# B&R Automation Studio project NAINV104C00R8L515F00 (part 32)

#### Act_InitLocal.st - Do Not Change!!!
```iecst
(** 2021-08-01 **)
ACTION Act_InitLocal:

	//Input Reference Link To Local Variable
	p_eAct ACCESS ADR(eAct);
	p_udiRstErr ACCESS ADR(udiRstErr);
	p_bPrep ACCESS ADR(bPrep);
	p_bEn ACCESS ADR(bEn);
	p_bDis ACCESS ADR(bDis);
	p_tyParam ACCESS ADR(tyParam);
	p_sIPAddr ACCESS ADR(sIPAddr);
	pa_usiMacAddr ACCESS ADR(a_usiMacAddr);
	p_tyDTStructure ACCESS ADR(tyDTStructure);
	p_dtCurrDT ACCESS ADR(dtCurrDT);
	p_sMcId ACCESS ADR(sMcId);
	p_sMagazineId ACCESS ADR(sMagazineId);
	p_iSlotId ACCESS ADR(iSlotId);
	p_eBoardTransfer1 ACCESS ADR(eBoardTransfer1);
	p_eBoardTransfer2 ACCESS ADR(eBoardTransfer2);
	p_eBoardTransfer3 ACCESS ADR(eBoardTransfer3);
	p_eBoardTransfer4 ACCESS ADR(eBoardTransfer4);
	p_sVersion ACCESS ADR(sVersion);
	p_sBarcode ACCESS ADR(sBarcode);
	p_sRecipeNm ACCESS ADR(sRecipeNm);
	p_udiSndBffrSize ACCESS ADR(udiSndBffrSize);
	p_udiRcvBffrSize ACCESS ADR(udiRcvBffrSize);
	p_udiAliveIdleTimeInSec ACCESS ADR(udiAliveIdleTimeInSec);
	p_tConnTimeOut ACCESS ADR(tConnTimeOut);
	p_diTransferInTO ACCESS ADR(diTransferInTO);
	p_bNewBrdAvlLastZone ACCESS ADR(bNewBrdAvl);
	p_bOpsRun ACCESS ADR(bOpsRun);
	p_udiFileKeepDay ACCESS ADR(udiFileKeepDay);
	p_sConfigFileName ACCESS ADR(sConfigFileName);
	p_sProgNm ACCESS ADR(sProgNm);
	p_bNtSettingsLoadDone ACCESS ADR(bNtSettingsLoadDone);
	p_bSvyPrep ACCESS ADR(bSvyPrep);
	p_bSvyEn ACCESS ADR(bSvyEn);
	p_bQueryWorkOrderInfo ACCESS ADR(bQueryWorkOrderInfo);
	p_bReinsertBrd ACCESS ADR(bReinsertBrd);
	p_tyHermesConfiguration ACCESS ADR(tyHermesCurrConfiguration);
	p_bUSHermesStopTransport1 ACCESS ADR(bUSHermesStopTransportSnd1); //Lane 1
	p_bUSHermesStopTransport2 ACCESS ADR(bUSHermesStopTransportSnd2); //Lane 2
	p_bUSHermesStopTransport3 ACCESS ADR(bUSHermesStopTransportSnd3); //Lane 3
	p_bUSHermesStopTransport4 ACCESS ADR(bUSHermesStopTransportSnd4); //Lane 4
	p_tyUSBoardArrived1 ACCESS ADR(tyUSHermesBoardArrivedData1); //Lane 1
	p_tyUSBoardArrived2 ACCESS ADR(tyUSHermesBoardArrivedData2); //Lane 2
	p_tyUSBoardArrived3 ACCESS ADR(tyUSHermesBoardArrivedData3); //Lane 3
	p_tyUSBoardArrived4 ACCESS ADR(tyUSHermesBoardArrivedData4); //Lane 4
	p_bDSHermesTransportFinished1 ACCESS ADR(bDSHermesTransportFinishedSnd1); //Lane 1
	p_bDSHermesTransportFinished2 ACCESS ADR(bDSHermesTransportFinishedSnd2); //Lane 2
	p_bDSHermesTransportFinished3 ACCESS ADR(bDSHermesTransportFinishedSnd3); //Lane 3
	p_bDSHermesTransportFinished4 ACCESS ADR(bDSHermesTransportFinishedSnd4); //Lane 4
	p_tyDSBoardDeparted1 ACCESS ADR(tyDSHermesBoardDepartedData1); //Lane 1
	p_tyDSBoardDeparted2 ACCESS ADR(tyDSHermesBoardDepartedData2); //Lane 2
	p_tyDSBoardDeparted3 ACCESS ADR(tyDSHermesBoardDepartedData3); //Lane 3
	p_tyDSBoardDeparted4 ACCESS ADR(tyDSHermesBoardDepartedData4); //Lane 4
	p_sInfoMsg ACCESS ADR(sInfoMsg);
	p_sInfoMsg1 ACCESS ADR(sInfoMsg1);
	p_sInfoMsg2 ACCESS ADR(sInfoMsg2);
	p_sInfoMsg3 ACCESS ADR(sInfoMsg3);
	p_sInfoMsg4 ACCESS ADR(sInfoMsg4);
	p_sInfoMsg5 ACCESS ADR(sInfoMsg5);
	p_sInfoMsg6 ACCESS ADR(sInfoMsg6);
	p_bInternalUse ACCESS ADR(bInternalUse);
	p_sInternalRcv ACCESS ADR(sInternalRcv);
	p_bAcceptCondition ACCESS ADR(bAcceptCondition);
	p_bAllZonesEmpty ACCESS ADR(bAllZonesEmpty);
	p_bDeleteWorkOrder ACCESS ADR(bDeleteWorkOrder);
	p_bFirstMcIntheLine ACCESS ADR(bFirstMcIntheLine);
	p_sRetainFileName ACCESS ADR(sRetainFileName);
	p_udiRetainDataAddr ACCESS ADR(udiRetainDataAddr);
	p_udiRetainDataLen ACCESS ADR(udiRetainDataLen);

END_ACTION
```

#### Act_Initial.st - Do Not Change!!!
```iecst
(** 2021-08-01 **)
ACTION Act_Initial:

	//Initial
	sStatTxt	:= a_sStatText[eStat];

	fbCreateSvr.udiSndBffrSize		:= p_udiSndBffrSize;
	fbCreateSvr.udiRcvBffrSize		:= p_udiRcvBffrSize;
	fbCreateSvr.udiAliveIdleTmInSec	:= p_udiAliveIdleTimeInSec;
	fbCreateSvr(bEn := FALSE);

	fbListen(bEn := FALSE);

	fbRcv.udiBffrSize	:= SIZEOF(sRcv);
	fbRcv.p_BffrDest	:= ADR(sRcv);
	fbRcv(bEn := FALSE);

	fbSend.p_BffrDest	:= ADR(sSnd);
	fbSend(bEn := FALSE);

	fbCloseSvr(bEn := FALSE);
	fbCloseClnt(bEn := FALSE);

	fbParseXMLTable.p_XMLTable	:= ADR(a_tyXMLTableDataRcv);

	fbCheckAlive(bEn := FALSE);

	fbCheckAliveSendPing(bEn := FALSE);

	fbCheckAliveRcvPing(bEn := FALSE);

	fbSequenceSvy.p_tyMsgTypeRcv	:= ADR(tyMsgTypeRcv);
	fbSequenceSvy(bEn := FALSE);

	fbSequenceTO(bEn := FALSE);

	fbFileAppend1.sDevice	:= 'Log';
	fbFileAppend1(bEn := FALSE);

	fbFileOldDel1.sDevice			:= 'Log';
	fbFileOldDel1.sPath				:= '';
	fbFileOldDel1.sKeyword			:= p_sProgNm;
	fbFileOldDel1.udiFileKeepDay	:= p_udiFileKeepDay;
	fbFileOldDel1(bEn := FALSE);

	fbFileRead1.sDevice			:= 'Retain';
	fbFileRead1.sFile			:= p_sRetainFileName;
	fbFileRead1.udiOffset		:= 0;
	fbFileRead1(bEn := FALSE);

	fbFileWrite1.sDevice		:= 'Retain';
	fbFileWrite1.sFile			:= p_sRetainFileName;
	fbFileWrite1.udiOffset		:= 0;
	fbFileWrite1.udiOption		:= 0;
	fbFileWrite1(bEn := FALSE);

END_ACTION
```

#### Act_Main.st - Do Not Change!!!
```iecst
(** 2021-08-01 **)
ACTION Act_Main:

	IF eStatOld <> eStat THEN
		fbFileOldDel1(bEn := FALSE);
		fbFileRead1(bEn := FALSE);
		fbFileWrite1(bEn := FALSE);
		bFileNotFound	:= FALSE;
		sStatTxt	:= a_sStatText[eStat];

		eStatOld	:= eStat;

		eStatus		:= Busy;
	END_IF

	//Main
	CASE eStat OF

		HermesActIdle:
			eStatus	:= Idle;

		HermesActBGStartRun:
			IF eStatus = Idle OR eStatus = Busy THEN

				bRun	:= TRUE;
				bStop	:= FALSE;
				eStatus	:= Done;

			END_IF

		HermesActBGStopRun:
			IF eStatus = Idle OR eStatus = Busy THEN

				bStop	:= TRUE;
				eStatus	:= Done;

			END_IF

		HermesActDeleteOldLog:
			IF eStatus = Idle OR eStatus = Busy THEN

				eStatus	:= Busy;

				fbFileOldDel1.dtDTNow	:= p_dtCurrDT;
				fbFileOldDel1(bEn := TRUE);
				IF fbFileOldDel1.udiStatus = 0 THEN
					eStatus	:= Done;
				ELSIF fbFileOldDel1.udiStatus < 65534 THEN
					eStatus		:= Error;

					IF fbFileOldDel1.udiStatus = 1910 THEN
						udiStatus	:= 10111;	//Get Directory Info Error While Deleting Old Log
					ELSIF fbFileOldDel1.udiStatus = 1911 THEN
						udiStatus	:= 10112;	//Directory Read Error While Deleting Old Log
					ELSIF fbFileOldDel1.udiStatus = 1912 THEN
						udiStatus	:= 10113;	//File Delete Error While Deleting Old Log
					ELSE
						udiStatus	:= fbFileOldDel1.udiStatus;
					END_IF
				END_IF

			END_IF

		HermesActReadRetain:
			IF eStatus = Idle OR eStatus = Busy THEN

				eStatus	:= Busy;

				fbFileRead1.p_Dest	:= p_udiRetainDataAddr;
				fbFileRead1.udiLen	:= p_udiRetainDataLen;
				fbFileRead1(bEn := TRUE);

				IF fbFileRead1.udiStatus = 0 THEN
					eStatus	:= Done;
				ELSIF fbFileRead1.udiStatus < 65534 THEN
					eStatus	:= Error;

					IF fbFileRead1.udiStatus = 1900 THEN
						udiStatus	:= 10114;	//File Open Error While Reading Retain File
					ELSIF fbFileRead1.udiStatus = 1902 THEN
						udiStatus	:= 10115;	//File Read Error While Reading Retain File
					ELSIF fbFileRead1.udiStatus = 1904 THEN
						udiStatus	:= 10116;	//File Close Error While Reading Retain File
					ELSIF fbFileRead1.udiStatus = 1915 THEN
						eStatus			:= Done;
						bFileNotFound	:= TRUE;
					ELSE
						udiStatus	:= fbFileRead1.udiStatus;
					END_IF
				END_IF

			END_IF

		HermesActWriteRetain:
			IF eStatus = Idle OR eStatus = Busy THEN

				eStatus	:= Busy;

				fbFileWrite1.p_Src	:= p_udiRetainDataAddr;
				fbFileWrite1.udiLen	:= p_udiRetainDataLen;
				fbFileWrite1(bEn := TRUE);

				IF fbFileWrite1.udiStatus = 0 THEN
					eStatus	:= Done;
				ELSIF fbFileWrite1.udiStatus < 65534 THEN
					eStatus	:= Error;

					IF fbFileWrite1.udiStatus = 1900 THEN
						udiStatus	:= 10117;	//File Open Error While Writing Retain File
					ELSIF fbFileWrite1.udiStatus = 1901 THEN
						udiStatus	:= 10118;	//File Create Error While Writing Retain File
					ELSIF fbFileWrite1.udiStatus = 1903 THEN
						udiStatus	:= 10119;	//File Write Error While Writing Retain File
					ELSIF fbFileWrite1.udiStatus = 1904 THEN
						udiStatus	:= 10120;	//File Close Error While Writing Retain File
					ELSIF fbFileWrite1.udiStatus = 1914 THEN
						udiStatus	:= 10121;	//Directory Does Not Exist While Writing Retain File
					ELSE
						udiStatus	:= fbFileWrite1.udiStatus;
					END_IF
				END_IF

			END_IF

		ELSE
			IF eStatus = Idle OR eStatus = Busy THEN
				eStatus	:= Done;
			END_IF

	END_CASE

END_ACTION
```

#### Act_Background.st - Do Not Change!!!
```iecst
(** 2021-08-01 **)
ACTION Act_Background:

	IF bRun = TRUE THEN
		IF udiSvrIdent = 0 THEN
			IF p_bInternalUse = FALSE THEN
				Act_Background_TCPCreateSvr;

				tyParamOld	:= p_tyParam;
			ELSE
				udiSvrIdent	:= 1;
			END_IF

		ELSE
			IF bRstConnection = FALSE THEN

				Act_Background_ChgConfig;

				IF udiClntIdent = 0 THEN
					IF p_bInternalUse = FALSE THEN
						Act_Background_TCPListen;
					ELSE
						udiClntIdent	:= 1;
					END_IF

				ELSE
					Act_Background_TCPRcv;

					Act_Background_NotificationRcv;

					Act_Background_IllegalMsg;
					Act_Background_ChkParamRcv;
					Act_Background_CmpParamRcv;
					Act_Background_UpdtConfig;

					IF bHandshakeDone = TRUE THEN
						IF (p_tyParam.tSndAlive <> T#0s) AND (p_tyParam.tRcvAlive <> T#0s) THEN
							IF tySServiceDescriptionRcv.tyData.tySupportedFeatures.bFeatureCheckAliveResponse = TRUE AND p_tyParam.bFeatureCheckAliveResponse = TRUE THEN
								Act_Background_ChkAliveSendPing;
								Act_Background_ChkAliveRcvPing;
							ELSE
								Act_Background_ChkAlive;
							END_IF
						ELSE
							fbCheckAlive(bEn := FALSE);
							fbCheckAliveSendPing(bEn := FALSE);
							fbCheckAliveRcvPing(bEn := FALSE);
						END_IF
					END_IF

					Act_Background_Sequence;
					Act_Background_SequenceTO;
					Act_Background_Err;

					IF tySServiceDescriptionRcv.tyAvl.tySupportedFeatures.bFeatureSendWorkOrderInfo = TRUE AND (p_tyParam.bFeatureQueryWorkOrderInfo OR p_bHermesReinsertBoard) AND bHandshakeDone THEN
						Act_Background_QueryWorkOrderInfo;
					END_IF

					Act_Background_SendBoardArrivedLane1;
					Act_Background_SendBoardArrivedLane2;
					Act_Background_SendBoardArrivedLane3;
					Act_Background_SendBoardArrivedLane4;
					Act_Background_SendBoardDepartedLane1;
					Act_Background_SendBoardDepartedLane2;
					Act_Background_SendBoardDepartedLane3;
					Act_Background_SendBoardDepartedLane4;
					Act_Background_TCPSend;

					Act_Background_Log;

				END_IF

			ELSE
				IF udiClntIdent <> 0 THEN
					Act_Background_TCPCloseClnt;
				ELSE
					IF udiSvrIdent <> 0 THEN
						Act_Background_TCPCloseSvr;
					END_IF
				END_IF

			END_IF

			//Second Client Connected
			IF udiClntIdentExtra = 0 THEN

			ELSE

			END_IF

		END_IF

		Act_Background_Stop;

	END_IF

	IF EDGENEG(bRun) OR EDGENEG(udiSvrIdent = 0) THEN
		//Reset
		fbCreateSvr(bEn := FALSE);
	END_IF

	IF EDGENEG(bRun) OR EDGENEG(udiClntIdent = 0) THEN
		//Reset
		fbListen(bEn := FALSE);

		bConnected	:= bRun;
	END_IF

	IF EDGENEG(bRun) OR EDGENEG(udiSvrIdent <> 0) OR EDGENEG(udiClntIdent <> 0) THEN
		fbRcv(bEn := FALSE);
		fbSequenceSvy(bEn := FALSE);
		fbSequenceTO(bEn := FALSE);
		fbCheckAlive(bEn := FALSE);
		fbCheckAliveSendPing(bEn := FALSE);
		fbCheckAliveRcvPing(bEn := FALSE);
		fbSend(bEn := FALSE);

		fbFileAppend1(bEn := FALSE);
		iWriteLogStep	:= 0;

		bConnected		:= FALSE;
		bHandshakeDone	:= FALSE;
		bRstState		:= FALSE;

		memset(ADR(tyMsgTypeRcv) , 0 , SIZEOF(tyMsgTypeRcv));
		memset(ADR(a_eMsgSend) , 0 , SIZEOF(a_eMsgSend));
		udiMsgSendBffr	:= 0;
	END_IF

	IF EDGENEG(bRun) OR EDGENEG(udiSvrIdent <> 0) THEN
		bRstConnection	:= FALSE;
		fbCloseSvr(bEn := FALSE);
	END_IF

	IF EDGENEG(bRun) OR EDGENEG(udiClntIdent <> 0) THEN
		fbCloseClnt(bEn := FALSE);
	END_IF

	//Reset Error
	IF (eStatus1 = Error) AND bRstErr THEN
		eStatus1	:= Idle;
		udiStatus1	:= 0;

		fbCreateSvr(bEn := FALSE);
		fbListen(bEn := FALSE);
		fbRcv(bEn := FALSE);
		fbSequenceSvy(bEn := FALSE);
		fbSend(bEn := FALSE);
		fbCloseSvr(bEn := FALSE);
		fbCloseClnt(bEn := FALSE);
		fbCheckAlive(bEn := FALSE);
		fbCheckAliveSendPing(bEn := FALSE);
		fbCheckAliveRcvPing(bEn := FALSE);
		fbSequenceTO(bEn := FALSE);

		fbFileAppend1(bEn := FALSE);
		iWriteLogStep	:= 0;

		bConnected		:= FALSE;
		bHandshakeDone	:= FALSE;
		bRstConnection	:= FALSE;
		bRstState		:= FALSE;

		memset(ADR(tyMsgTypeRcv) , 0 , SIZEOF(tyMsgTypeRcv));
		memset(ADR(a_eMsgSend) , 0 , SIZEOF(a_eMsgSend));
		udiMsgSendBffr	:= 0;
	END_IF

	IF (eStatus2 = Error) AND bRstErr THEN
		eStatus2	:= Idle;
		udiStatus2	:= 0;

		fbSequenceTO(bEn := FALSE);

	END_IF

	IF (eStatus3 = Error) AND bRstErr THEN
		eStatus3	:= Idle;
		udiStatus3	:= 0;

		fbFileAppend1(bEn := FALSE);
		iWriteLogStep	:= 0;
	END_IF

END_ACTION
```

#### Act_Background_ProcessData.st - Do Not Change!!!
```iecst
(** 2021-08-01 **)
ACTION Act_Background_ProcessData:

	//Write Config into "Hermes"
	fbDelayTm(IN := bWriteConfig, PT := T#0.5S); //Small Delay 0.5s to let Hermes take the Data, before WriteConfig

	IF fbDelayTm.Q THEN

		eHermesAct := HermesActWriteConfig;
		eMcParamAct := McParamActWrite;

		IF p_eHermesStatus = Done AND p_eHermesStat = HermesActWriteConfig AND p_eMcParamStat = McParamActWrite AND p_eMcParamStatus = Done THEN

		eMcParamAct     := McParamActIdle;
	   	eHermesAct		:= HermesActIdle;
		bWriteConfig    := FALSE;
		bUpdateUIData   := TRUE;
		fbDelayTm(IN := FALSE);
		tyInfoData.sProgNm		:= p_sProgNm;
		tyInfoData.udiCode		:= 10000;
		tyInfoData.eSeverity	:= AlmSeverityInfo;
		tyInfoData.sAlmMsg		:= p_sInfoMsg;

	    ELSIF  (p_eHermesStatus = Error AND p_eHermesStat = HermesActWriteConfig) OR (p_eMcParamStat = McParamActWrite AND p_eMcParamStatus = Error)  THEN

			eMcParamAct     := McParamActIdle;
		    eHermesAct		:= HermesActIdle;
		    bWriteConfig    := FALSE;
		    bUpdateUIData   := FALSE;
			fbDelayTm(IN := FALSE);

			fHermesAddOneMsgSend(ADR(a_eMsgSend) , ADR(udiMsgSendBffr) , HermesMsgTypeNotification);

			udiStatus2 := 10199; //SetConfiguration Failed, Please Send Again
			tyNotificationSnd.tyAvl.bSeverity			:= TRUE;
			tyNotificationSnd.tyAvl.bNotificationCode	:= TRUE;
			tyNotificationSnd.tyAvl.bDescription		:= TRUE;
			tyNotificationSnd.tyData.eSeverity			:= HermesSeverityFatalError;
			tyNotificationSnd.tyData.iNotificationCode	:= UDINT_TO_INT(udiStatus2);
			tyNotificationSnd.tyData.sDescription		:= a_tyAlmText[udiStatus2].sAlmText;

		END_IF
	END_IF

	//Update UI
	IF bUpdateUIData THEN
		tyInfoData.sProgNm		:= p_sProgNm;
		tyInfoData.udiCode		:= 10000;
		tyInfoData.eSeverity	:= AlmSeverityInfo;
		tyInfoData.sAlmMsg		:= p_sInfoMsg;
	END_IF

	//Auto Reset
	fbDelayTm1(IN := bUpdateUIData , PT := T#2S); //Auto reset the Info Msg C0009 page. No need press.
	IF fbDelayTm1.Q = TRUE THEN

		//Clear Info Message
		tyInfoData.sProgNm		:= '';
		tyInfoData.udiCode		:= 0;
		tyInfoData.eSeverity	:= AlmSeverityNA;
		tyInfoData.sAlmMsg		:= '';

		bUpdateUIData  := FALSE;
		bFoundIndexUS1 := FALSE;
		bFoundIndexUS2 := FALSE;
		bFoundIndexUS3 := FALSE;
		bFoundIndexUS4 := FALSE;
		bFoundIndexDS1 := FALSE;
		bFoundIndexDS2 := FALSE;
		bFoundIndexDS3 := FALSE;
		bFoundIndexDS4 := FALSE;

		fbDelayTm1(IN := FALSE);
	END_IF

	//BatchId from Supervisory System
	sBatchId := tySendWorkOrderInfoAcc.tyData.sBatchId;

	//Retain sWorkOrderId for machine power cycle
	p_udiRetainDataAddr	:= ADR(sWorkOrderId);
	p_udiRetainDataLen	:= SIZEOF(sWorkOrderId);

	//Write Retain
	IF EDGEPOS(bRcvWorkOrderInfo1) THEN
    	sWorkOrderId := tySendWorkOrderInfoAcc.tyData.sWorkOrderId; //Receive from Svy
		p_eAct := HermesActWriteRetain;

	ELSIF EDGENEG(p_bSvyEn = TRUE) OR EDGENEG(p_bSvyPrep = TRUE) THEN
		sWorkOrderId := ''; //Empty if Supervisory Hermes disable
		p_eAct := HermesActWriteRetain;

	ELSIF EDGENEG(p_tyHermesConfiguration.tySvyParam.bFeatureQueryWorkOrderInfo = TRUE) THEN
		sWorkOrderId := ''; //Empty if no support
		p_eAct := HermesActWriteRetain;

	ELSIF EDGEPOS(p_bDeleteWorkOrder) THEN
		sWorkOrderId := ''; //Delete from UI
		p_eAct := HermesActWriteRetain;
		p_bDeleteWorkOrder := FALSE;
	END_IF

	IF eStatus = Done AND eStat = HermesActWriteRetain THEN
		p_eAct		:= HermesActIdle;
	END_IF

//	//Testing -> Read Retain
//	IF EDGEPOS(bTest) THEN
//		p_eAct := HermesActReadRetain;
//	END_IF
//
//	IF eStatus = Done AND eStat = HermesActReadRetain THEN
//		p_eAct		:= HermesActIdle;
//	END_IF

	IF EDGEPOS(bTest) THEN

	END_IF

END_ACTION
```

#### Act_Background_TCPCreateSvr.st - Do Not Change!!!
```iecst
(** 2021-08-01 **)
ACTION Act_Background_TCPCreateSvr:

	IF eStatus1 <> Error THEN

		//Create Server
		fbCreateSvr.sSvrIP				:= p_sIPAddr;
		fbCreateSvr.uiSvrPort			:= p_tyParam.uiSvySvstemPort;
		fbCreateSvr(bEn := TRUE);

		IF fbCreateSvr.udiStatus = 0 THEN
			udiSvrIdent	:= fbCreateSvr.udiTCPIdent;
			fbCreateSvr(bEn := FALSE);

		ELSIF fbCreateSvr.udiStatus < 65534 THEN
			eStatus1	:= Error;

			IF fbCreateSvr.udiStatus = 2300 THEN
				udiStatus1	:= 10000;	//Invalid Ident While Creating Server
			ELSIF fbCreateSvr.udiStatus = 2302 THEN
				udiStatus1	:= 10001;	//Setting Keep Alive Interval Time Error While Creating Server
			ELSIF fbCreateSvr.udiStatus = 2303 THEN
				udiStatus1	:= 10002;	//Setting Keep Alive Idle Time Error While Creating Server
			ELSIF fbCreateSvr.udiStatus = 2304 THEN
				udiStatus1	:= 10003;	//Setting Keep Alive Count Error While Creating Server
			ELSIF fbCreateSvr.udiStatus = 2305 THEN
				udiStatus1	:= 10004;	//Setting Keep Alive Error While Creating Server
			ELSIF fbCreateSvr.udiStatus = 2306 THEN
				udiStatus1	:= 10005;	//Setting Receive Buffer Error While Creating Server
			ELSIF fbCreateSvr.udiStatus = 2307 THEN
				udiStatus1	:= 10006;	//Setting Send Buffer Error While Creating Server
			ELSIF fbCreateSvr.udiStatus = 2308 THEN
				udiStatus1	:= 10007;	//Setting No Waiting Error While Creating Server
			ELSIF fbCreateSvr.udiStatus = 2309 THEN
				udiStatus1	:= 10008;	//TCP Open Port Error While Creating Server
			ELSIF fbCreateSvr.udiStatus = 2310 THEN
				udiStatus1	:= 10009;	//Closing TCP Error While Creating Server
			ELSE
				udiStatus1	:= fbCreateSvr.udiStatus;
			END_IF

		END_IF

	END_IF

END_ACTION
```

#### Act_Background_TCPListen.st - Do Not Change!!!
```iecst
(** 2021-08-01 **)
ACTION Act_Background_TCPListen:

	IF eStatus1 <> Error AND eStatus2 <> Error THEN

		fbListen.udiSvrIdent	:= udiSvrIdent;
		fbListen(bEn := TRUE);

		IF fbListen.udiStatus = 0 THEN
			udiClntIdent	:= fbListen.udiClntIdent;
			fbListen(bEn := FALSE);

		ELSIF fbListen.udiStatus = 2311 THEN //No Client Connected
			fbListen(bEn := FALSE);

		ELSIF fbListen.udiStatus = 2312 OR (bConnected=FALSE) THEN
			udiStatus4	:= 10012;	//Supervisory Hermes Connection Lost
			fbListen(bEn := FALSE); //add

		ELSIF fbListen.udiStatus < 65534 THEN
			eStatus1	:= Error;

			IF fbListen.udiStatus = 2300 THEN
				udiStatus1	:= 10010;	//Invalid Ident While Listening Client
			ELSE
				udiStatus1	:= fbListen.udiStatus;
			END_IF

		END_IF

	END_IF

END_ACTION
```

#### Act_Background_TCPRcv.st - Do Not Change!!!
```iecst
(** 2020-10-20 **)
ACTION Act_Background_TCPRcv:

	IF eStatus1 <> Error THEN

		//Receive Data
		IF p_bInternalUse = FALSE THEN
			fbRcv.udiTCPIdent	:= udiClntIdent;
			fbRcv(bEn := TRUE);
		ELSE
			sRcv	:= p_sInternalRcv;
		END_IF

		IF (fbRcv.udiStatus = 0) OR ((p_bInternalUse = TRUE) AND (LEN(sRcv) > 0)) THEN

			fLogDTConvert(ADR(sDT) , p_dtCurrDT);
			memset(ADR(a_sLogList[udiLogCntr]) , 0 , SIZEOF(a_sLogList[udiLogCntr]));
			memcpy(ADR(a_sLogList[udiLogCntr]) + LEN(a_sLogList[udiLogCntr]) , ADR(sDT) , LEN(sDT));
			memcpy(ADR(a_sLogList[udiLogCntr]) + LEN(a_sLogList[udiLogCntr]) , ADR('$r$n') , LEN('$r$n'));
			memcpy(ADR(a_sLogList[udiLogCntr]) + LEN(a_sLogList[udiLogCntr]) , ADR('RCV_FRM_SVY$r$n') , LEN('RCV_FRM_SVY$r$n'));
			memcpy(ADR(a_sLogList[udiLogCntr]) + LEN(a_sLogList[udiLogCntr]) , ADR(sRcv) , LEN(sRcv));
			memcpy(ADR(a_sLogList[udiLogCntr]) + LEN(a_sLogList[udiLogCntr]) , ADR('$r$n$r$n') , LEN('$r$n$r$n'));

			udiLogCntr	:= udiLogCntr + 1;
			IF udiLogCntr = 11 THEN
				udiLogCntr	:= 1;
			END_IF

			fXMLConvertToTable(ADR(sRcv) , LEN(sRcv) , ADR(a_tyXMLTableDataRcv) , ADR(a_tyXMLTableDataRcv[0].sTitle) , SIZEOF(a_tyXMLTableDataRcv[0].sTitle) , ADR(a_tyXMLTableDataRcv[0].sValue) , SIZEOF(a_tyXMLTableDataRcv[0].sValue) , ADR(a_tyXMLTableDataRcv[0].uiSize) , SIZEOF(a_tyXMLTableDataRcv[0]) , SIZEOF(a_tyXMLTableDataRcv) / SIZEOF(a_tyXMLTableDataRcv[0]) , ADR(udiXMLTableWriteIdx));

			fbParseXMLTable.iTotalIdxWrite	:= UDINT_TO_INT(udiXMLTableWriteIdx);
			fbParseXMLTable;

			IF fbParseXMLTable.tyMsgType.bCheckAlive = TRUE THEN
				tyMsgTypeRcv.bCheckAlive	:= TRUE;
				tyCheckAliveRcv				:= fbParseXMLTable.tyCheckAlive;
			END_IF

			IF fbParseXMLTable.tyMsgType.bCheckAlivePing = TRUE THEN
				tyMsgTypeRcv.bCheckAlivePing	:= TRUE;
				tyCheckAlivePingRcv				:= fbParseXMLTable.tyCheckAlivePing;
			END_IF

			IF fbParseXMLTable.tyMsgType.bCheckAlivePong = TRUE THEN
				tyMsgTypeRcv.bCheckAlivePong	:= TRUE;
				tyCheckAlivePongRcv				:= fbParseXMLTable.tyCheckAlivePong;
			END_IF

			IF fbParseXMLTable.tyMsgType.bServiceDescription = TRUE THEN
				tyMsgTypeRcv.bServiceDescription	:= TRUE;
				tyServiceDescriptionRcv				:= fbParseXMLTable.tyServiceDescription;
			END_IF

			IF fbParseXMLTable.tyMsgType.bSServiceDescription = TRUE THEN
				tyMsgTypeRcv.bSServiceDescription	    := TRUE;
				tySServiceDescriptionRcv				:= fbParseXMLTable.tySServiceDescription;
			END_IF

			IF fbParseXMLTable.tyMsgType.bNotification = TRUE THEN
				tyMsgTypeRcv.bNotification	:= TRUE;
				tyNotificationRcv			:= fbParseXMLTable.tyNotification;
			END_IF

			IF fbParseXMLTable.tyMsgType.bBoardAvailable = TRUE THEN
				tyMsgTypeRcv.bBoardAvailable	:= TRUE;
				tyBoardAvailableRcv				:= fbParseXMLTable.tyBoardAvailable;

			END_IF

			IF fbParseXMLTable.tyMsgType.bRevokeBoardAvailable = TRUE THEN
				tyMsgTypeRcv.bRevokeBoardAvailable	:= TRUE;
			END_IF

			IF fbParseXMLTable.tyMsgType.bMachineReady = TRUE THEN
				tyMsgTypeRcv.bMachineReady	:= TRUE;
				tyMachineReady				:= fbParseXMLTable.tyMachineReady;
			END_IF

			IF fbParseXMLTable.tyMsgType.bRevokeMachineReady = TRUE THEN
				tyMsgTypeRcv.bRevokeMachineReady	:= TRUE;
			END_IF

			IF fbParseXMLTable.tyMsgType.bStartTransport = TRUE THEN
				tyMsgTypeRcv.bStartTransport	:= TRUE;
				tyStartTransport				:= fbParseXMLTable.tyStartTransport;
			END_IF

			IF fbParseXMLTable.tyMsgType.bStopTransport = TRUE THEN
				tyMsgTypeRcv.bStopTransport	:= TRUE;
				tyStopTransport				:= fbParseXMLTable.tyStopTransport;
			END_IF

			IF fbParseXMLTable.tyMsgType.bTransportFinished = TRUE THEN
				tyMsgTypeRcv.bTransportFinished	:= TRUE;
				tyTransportFinished				:= fbParseXMLTable.tyTransportFinished;
			END_IF

			IF fbParseXMLTable.tyMsgType.bSetConfiguration = TRUE THEN
				tyMsgTypeRcv.bSetConfiguration	:= TRUE;
				tySetConfigurationRcv			:= fbParseXMLTable.tySetConfiguration;
			END_IF

			IF fbParseXMLTable.tyMsgType.bGetConfiguration = TRUE THEN
				tyMsgTypeRcv.bGetConfiguration	:= TRUE;
			END_IF

			IF fbParseXMLTable.tyMsgType.bCurrentConfiguration = TRUE THEN
				tyMsgTypeRcv.bCurrentConfiguration	:= TRUE;
				tyCurrentConfigurationRcv			:= fbParseXMLTable.tyCurrentConfiguration;
			END_IF

			IF fbParseXMLTable.tyMsgType.bBoardForecast = TRUE THEN
				tyMsgTypeRcv.bBoardForecast	:= TRUE;
				tyBoardForecast				:= fbParseXMLTable.tyBoardForecast;
			END_IF

			IF fbParseXMLTable.tyMsgType.bBoardArrived = TRUE THEN
				tyMsgTypeRcv.bBoardArrived	:= TRUE;
				tyBoardArrivedRcv				:= fbParseXMLTable.tyBoardArrived;
			END_IF

			IF fbParseXMLTable.tyMsgType.bBoardDeparted = TRUE THEN
				tyMsgTypeRcv.bBoardDeparted	:= TRUE;
				tyBoardDepartedRcv				:= fbParseXMLTable.tyBoardDeparted;
			END_IF

			IF fbParseXMLTable.tyMsgType.bQueryBoardInfo = TRUE THEN
				tyMsgTypeRcv.bQueryBoardInfo	:= TRUE;
				tyQueryBoardInfo				:= fbParseXMLTable.tyQueryBoardInfo;
			END_IF

			IF fbParseXMLTable.tyMsgType.bSendBoardInfo = TRUE THEN
				tyMsgTypeRcv.bSendBoardInfo	    := TRUE;
				tySendBoardInfo				    := fbParseXMLTable.tySendBoardInfo;
			END_IF

			IF fbParseXMLTable.tyMsgType.bQueryWorkOrderInfo = TRUE THEN
				tyMsgTypeRcv.bQueryWorkOrderInfo	:= TRUE;
				tyQueryWorkOrderInfo				:= fbParseXMLTable.tyQueryWorkOrderInfo;
			END_IF

			IF fbParseXMLTable.tyMsgType.bSendWorkOrderInfo = TRUE THEN
				tyMsgTypeRcv.bSendWorkOrderInfo	    := TRUE;
				tySendWorkOrderInfoRcv			    := fbParseXMLTable.tySendWorkOrderInfo;
			END_IF

			fbRcv(bEn := FALSE);

			memset(ADR(sRcv) , 0 , SIZEOF(sRcv));

		ELSIF (fbRcv.udiStatus = 2317) AND (p_bInternalUse = FALSE) THEN
			fbRcv(bEn := FALSE);

			memset(ADR(sRcv) , 0 , SIZEOF(sRcv));

		ELSIF (fbRcv.udiStatus = 2316) AND (p_bInternalUse = FALSE) THEN
			bRstConnection	:= TRUE;

			memset(ADR(sRcv) , 0 , SIZEOF(sRcv));

		ELSIF (fbRcv.udiStatus = 2318) AND (p_bInternalUse = FALSE) THEN
			bRstConnection	:= TRUE;

			memset(ADR(sRcv) , 0 , SIZEOF(sRcv));

		ELSIF (fbRcv.udiStatus < 65534) AND (p_bInternalUse = FALSE) THEN
			eStatus1	:= Error;

			IF fbRcv.udiStatus = 2300 THEN
				udiStatus1	:= 10014;	//Invalid Ident While Receiving Data
			ELSIF fbRcv.udiStatus = 2319 THEN
				udiStatus1	:= 10015;	//TCP Receive Data Error While Receiving Data
			ELSE
				udiStatus1	:= fbRcv.udiStatus;
			END_IF

			memset(ADR(sRcv) , 0 , SIZEOF(sRcv));

		END_IF

	END_IF

END_ACTION
```

#### Act_Background_IllegalMsg.st - Do Not Change!!!
```iecst
(** 2021-08-01 **)
ACTION Act_Background_IllegalMsg:

	IF eStatus2 <> Error THEN

		udiStatus2	:= fHermesIllegalMsgSvy(fbSequenceSvy.eState , tyMsgTypeRcv);

		IF udiStatus2 <> 0 THEN
			eStatus2	:= Error;

			IF udiStatus2 = 2940 THEN
				udiStatus2	:= 10016;	//Receive SetConfiguration While Supervisory In Not Connected State
			ELSIF udiStatus2 = 2941 THEN
				udiStatus2	:= 10017;	//Receive GetConfiguration While Supervisory In Not Connected State
			ELSIF udiStatus2 = 2942 THEN
				udiStatus2	:= 10018;	//Receive CurrConfiguration While Supervisory In Not Connected State
			ELSIF udiStatus2 = 2943 THEN
				udiStatus2	:= 10019;	//Receive SendWorkOrderInfo While Supervisory In Not Connected State
			ELSIF udiStatus2 = 2944 THEN
				udiStatus2	:= 10020;	//Receive QueryWorkOrderInfo While Supervisory In Not Connected State
			ELSIF udiStatus2 = 2945 THEN
				udiStatus2	:= 10021;	//Receive BoardArrived While Supervisory In Not Connected State
			ELSIF udiStatus2 = 2946 THEN
				udiStatus2	:= 10022;	//Receive BoardDeparted While Supervisory In Not Connected State
			ELSIF udiStatus2 = 2947 THEN
				udiStatus2	:= 10023;
			ELSIF udiStatus2 = 2948 THEN
				udiStatus2	:= 10024;
			ELSIF udiStatus2 = 2949 THEN
				udiStatus2	:= 10025;
			ELSIF udiStatus2 = 2950 THEN
				udiStatus2	:= 10026;
			ELSIF udiStatus2 = 2951 THEN
				udiStatus2	:= 10027;	//Receive Supervisory ServiceDescription While Supervisory In Service Description State
			ELSIF udiStatus2 = 2952 THEN
				udiStatus2	:= 10028;	//Receive SetConfiguration While Supervisory In Service Description State
			ELSIF udiStatus2 = 2953 THEN
				udiStatus2	:= 10029;	//Receive GetConfiguration While Supervisory In Service Description State
			ELSIF udiStatus2 = 2954 THEN
				udiStatus2	:= 10030;	//Receive CurrConfiguration While Supervisory In Service Description State
			ELSIF udiStatus2 = 2955 THEN
				udiStatus2	:= 10031;	//Receive SendWorkOrderInfo While Supervisory In Service Description State
			ELSIF udiStatus2 = 2956 THEN
				udiStatus2	:= 10032;	//Receive QueryWorkOrderInfo While Supervisory In Service Description State
			ELSIF udiStatus2 = 2957 THEN
				udiStatus2	:= 10033;	//Receive BoardArrived While Supervisory In Service Description State
			ELSIF udiStatus2 = 2958 THEN
				udiStatus2	:= 10034;	//Receive BoardDeparted While Supervisory In Service Description State
			ELSIF udiStatus2 = 2959 THEN
				udiStatus2	:= 10035;
			ELSIF udiStatus2 = 2960 THEN
				udiStatus2	:= 10036;
			ELSIF udiStatus2 = 2961 THEN
				udiStatus2	:= 10037;
			ELSIF udiStatus2 = 2962 THEN
				udiStatus2	:= 10038;
			ELSIF udiStatus2 = 2963 THEN
				udiStatus2	:= 10039;	//Receive Supervisory ServiceDescription While Supervisory In Connected State
			ELSIF udiStatus2 = 2964 THEN
				udiStatus2	:= 10040;	//Receive CurrConfiguration While Supervisory In Connected State
			ELSIF udiStatus2 = 2965 THEN
				udiStatus2	:= 10041;	//Receive QueryWorkOrderInfo While Supervisory In Connected State
			ELSIF udiStatus2 = 2966 THEN
				udiStatus2	:= 10042;	//Receive BoardArrived While Supervisory In Connected State
			ELSIF udiStatus2 = 2967 THEN
				udiStatus2	:= 10043;	//Receive BoardDeparted While Supervisory In Connected State
			ELSIF udiStatus2 = 2968 THEN
				udiStatus2	:= 10044;
			ELSIF udiStatus2 = 2969 THEN
				udiStatus2	:= 10045;
			ELSIF udiStatus2 = 2970 THEN
				udiStatus2	:= 10046;
			ELSIF udiStatus2 = 2971 THEN
				udiStatus2	:= 10047;
			END_IF

			fHermesAddOneMsgSend(ADR(a_eMsgSend) , ADR(udiMsgSendBffr) , HermesMsgTypeNotification);

			tyNotificationSnd.tyAvl.bSeverity			:= TRUE;
			tyNotificationSnd.tyAvl.bNotificationCode	:= TRUE;
			tyNotificationSnd.tyAvl.bDescription		:= TRUE;
			tyNotificationSnd.tyData.eSeverity			:= HermesSeverityFatalError;
			tyNotificationSnd.tyData.iNotificationCode	:= UDINT_TO_INT(udiStatus2);
			tyNotificationSnd.tyData.sDescription		:= a_tyAlmText[udiStatus2].sAlmText;

		END_IF

	END_IF

END_ACTION
```

#### Act_Background_ChkParamRcv.st - Do Not Change!!!
```iecst
(** 2021-08-01 **)
ACTION Act_Background_ChkParamRcv:

	IF eStatus2 <> Error THEN

		//Check Parameter Receive
		IF tyMsgTypeRcv.bSServiceDescription = TRUE THEN
			udiStatus2	:= fHermesChkParamSSD(tySServiceDescriptionRcv);

			IF udiStatus2 = 2731 THEN
				udiStatus2	:= 0;
			END_IF

			IF udiStatus2 <> 0 THEN
				eStatus2	:= Error;

				IF udiStatus2 = 2719 THEN
					udiStatus2	:= 10087;	//SystemId Missing While Checking Service Description
               	ELSIF udiStatus2 = 2730 THEN
					udiStatus2	:= 10088;	//Version Missing While Checking Service Description
				ELSIF udiStatus2 = 2731 THEN
					udiStatus2	:= 10089;	//SupportedFeatures Missing While Checking Service Description
				END_IF

				fHermesAddOneMsgSend(ADR(a_eMsgSend) , ADR(udiMsgSendBffr) , HermesMsgTypeNotification);

				tyNotificationSnd.tyAvl.bSeverity			:= TRUE;
				tyNotificationSnd.tyAvl.bNotificationCode	:= TRUE;
				tyNotificationSnd.tyAvl.bDescription		:= TRUE;
				tyNotificationSnd.tyData.eSeverity			:= HermesSeverityFatalError;
				tyNotificationSnd.tyData.iNotificationCode	:= UDINT_TO_INT(udiStatus2);
				tyNotificationSnd.tyData.sDescription		:= a_tyAlmText[udiStatus2].sAlmText;

			END_IF
		END_IF

		IF tyMsgTypeRcv.bNotification = TRUE THEN
			udiStatus2	:= fHermesChkParamN(tyNotificationRcv);

			IF udiStatus2 <> 0 THEN
				eStatus2	:= Error;

				IF udiStatus2 = 2732 THEN
					udiStatus2	:= 10092;	//NotificationCode Out Of Range While Checking Notification
				ELSIF udiStatus2 = 2733 THEN
					udiStatus2	:= 10093;	//NotificationCode Missing While Checking Notification
				ELSIF udiStatus2 = 2734 THEN
					udiStatus2	:= 10094;	//Severity Missing While Checking Notification
				ELSIF udiStatus2 = 2735 THEN
					udiStatus2	:= 10095;	//Description Missing While Checking Notification
				END_IF

				fHermesAddOneMsgSend(ADR(a_eMsgSend) , ADR(udiMsgSendBffr) , HermesMsgTypeNotification);

				tyNotificationSnd.tyAvl.bSeverity			:= TRUE;
				tyNotificationSnd.tyAvl.bNotificationCode	:= TRUE;
				tyNotificationSnd.tyAvl.bDescription		:= TRUE;
				tyNotificationSnd.tyData.eSeverity			:= HermesSeverityFatalError;
				tyNotificationSnd.tyData.iNotificationCode	:= UDINT_TO_INT(udiStatus2);
				tyNotificationSnd.tyData.sDescription		:= a_tyAlmText[udiStatus2].sAlmText;

			END_IF
		END_IF

	END_IF

END_ACTION
```

#### Act_Background_CmpParamRcv.st - Do Not Change!!!
```iecst
(** 2021-08-01 **)
ACTION Act_Background_CmpParamRcv:

	IF eStatus2 <> Error THEN

		IF tySServiceDescriptionRcv.tyAvl.tySupportedFeatures.bFeatureSendWorkOrderInfo = TRUE AND p_tyParam.bFeatureQueryWorkOrderInfo THEN

			IF tyMsgTypeRcv.bSendWorkOrderInfo = TRUE AND (p_bQueryWorkOrderInfo OR p_bReinsertBrd) THEN	//Hermes 1.3 Board Reinsert Function
				udiStatus2	:= fHermesChkParamSWQW(tySendWorkOrderInfoRcv , tyQueryWorkOrderInfo);

				IF udiStatus2 <> 0 THEN
					eStatus2	:= Error;

					IF udiStatus2 = 2767 THEN
						udiStatus2	:= 10164;	//QueryId Mismatch While Checking SendWorkOrderId & QueryWorkOrderId
					ELSIF udiStatus2 = 2768 THEN
						udiStatus2	:= 10165;	//QueryId Missing While Checking SendWorkOrderId & QueryWorkOrderId
					END_IF

					fHermesAddOneMsgSend(ADR(a_eMsgSend) , ADR(udiMsgSendBffr) , HermesMsgTypeNotification);

					tyNotificationSnd.tyAvl.bSeverity			:= TRUE;
					tyNotificationSnd.tyAvl.bNotificationCode	:= TRUE;
					tyNotificationSnd.tyAvl.bDescription		:= TRUE;
					tyNotificationSnd.tyData.eSeverity			:= HermesSeverityError;
					tyNotificationSnd.tyData.iNotificationCode	:= UDINT_TO_INT(udiStatus2);
					tyNotificationSnd.tyData.sDescription		:= a_tyAlmText[udiStatus2].sAlmText;

					tyMsgTypeRcv.bSendWorkOrderInfo := FALSE; //reset, else latching
				END_IF
			END_IF
		END_IF

	END_IF

END_ACTION
```

#### Act_Background_Sequence.st - Do Not Change!!!
```iecst
(** 2021-08-01 **)
ACTION Act_Background_Sequence:

	IF eStatus1 <> Error THEN

		//Sequence
		fbSequenceSvy.bRstState		        := bRstState;
		fbSequenceSvy(bEn := TRUE);

		IF fbSequenceSvy.eState >= HermesStateConnected THEN
			bHandshakeDone	:= TRUE;
		ELSE
			bHandshakeDone	:= FALSE;
		END_IF

		IF fbSequenceSvy.eMsgTypeSnd = HermesMsgTypeSServiceDescription THEN
			fHermesAddOneMsgSend(ADR(a_eMsgSend) , ADR(udiMsgSendBffr) , HermesMsgTypeSServiceDescription);

			tySServiceDescriptionSnd.tyData.sSystemId									        := p_sMcId;
			tySServiceDescriptionSnd.tyData.sVersion											:= p_sVersion;
			tySServiceDescriptionSnd.tyData.tySupportedFeatures.bFeatureCheckAliveResponse   	:= (p_tyParam.bFeatureCheckAliveResponse) AND (p_tyParam.tRcvAlive <> T#0s) AND (p_tyParam.tSndAlive <> T#0s);
			tySServiceDescriptionSnd.tyData.tySupportedFeatures.bFeatureConfiguration	    	:= p_tyParam.bFeatureConfiguration;
			tySServiceDescriptionSnd.tyData.tySupportedFeatures.bFeatureBoardTracking	    	:= p_tyParam.bFeatureBoardTracking;
			tySServiceDescriptionSnd.tyData.tySupportedFeatures.bFeatureQueryWorkOrderInfo	    := p_tyParam.bFeatureQueryWorkOrderInfo;
			tySServiceDescriptionSnd.tyData.tySupportedFeatures.bFeatureSendWorkOrderInfo    	:= FALSE; //p_tyParam.bFeatureSendWorkOrderInfo

			tySServiceDescriptionSnd.tyAvl.bSystemId										    := tySServiceDescriptionSnd.tyData.sSystemId<>'';
			tySServiceDescriptionSnd.tyAvl.bVersion											    := TRUE;
			tySServiceDescriptionSnd.tyAvl.bSupportedFeatures								    := p_tyParam.bFeatureCheckAliveResponse OR p_tyParam.bFeatureConfiguration OR p_tyParam.bFeatureBoardTracking OR p_tyParam.bFeatureQueryWorkOrderInfo OR p_tyParam.bFeatureSendWorkOrderInfo;
			tySServiceDescriptionSnd.tyAvl.tySupportedFeatures.bFeatureCheckAliveResponse	    := (p_tyParam.bFeatureCheckAliveResponse) AND (p_tyParam.tRcvAlive <> T#0s) AND (p_tyParam.tSndAlive <> T#0s);
			tySServiceDescriptionSnd.tyAvl.tySupportedFeatures.bFeatureConfiguration			:= p_tyParam.bFeatureConfiguration;
			tySServiceDescriptionSnd.tyAvl.tySupportedFeatures.bFeatureBoardTracking	        := p_tyParam.bFeatureBoardTracking;
			tySServiceDescriptionSnd.tyAvl.tySupportedFeatures.bFeatureQueryWorkOrderInfo		:= p_tyParam.bFeatureQueryWorkOrderInfo;
			tySServiceDescriptionSnd.tyAvl.tySupportedFeatures.bFeatureSendWorkOrderInfo    	:= FALSE; //p_tyParam.bFeatureSendWorkOrderInfo

		ELSIF fbSequenceSvy.eMsgTypeSnd = HermesMsgTypeCurrConfiguration AND bWriteConfig = FALSE AND bUpdateUIData = FALSE THEN
			fHermesAddOneMsgSend(ADR(a_eMsgSend) , ADR(udiMsgSendBffr) , HermesMsgTypeCurrConfiguration);

			tyCurrentConfigurationSnd.tyData.sMachineId			                        		        := p_sMcId;
			tyCurrentConfigurationSnd.tyData.uiSupervisorySystemPort	                             	:= p_tyHermesConfiguration.tySvyParam.uiSvySvstemPort;
			tyCurrentConfigurationSnd.tyData.a_tyUpstreamConfigurations[0].iUpstreamLaneId	            := p_tyHermesConfiguration.a_tyUSParam[0].iLaneID;
			tyCurrentConfigurationSnd.tyData.a_tyUpstreamConfigurations[0].sHostAddress	                := p_tyHermesConfiguration.a_tyUSParam[0].sHostAddress;
			tyCurrentConfigurationSnd.tyData.a_tyUpstreamConfigurations[0].sUpstreamInterfaceId        	:= p_tyHermesConfiguration.a_tyUSParam[0].sUpstreamInterfaceId;
			tyCurrentConfigurationSnd.tyData.a_tyUpstreamConfigurations[0].uiPort                      	:= p_tyHermesConfiguration.a_tyUSParam[0].uiHostPort;

			tyCurrentConfigurationSnd.tyData.a_tyDownstreamConfigurations[0].iDownstreamLaneId	        := p_tyHermesConfiguration.a_tyDSParam[0].iLaneID;
			tyCurrentConfigurationSnd.tyData.a_tyDownstreamConfigurations[0].sClientAddress	            := p_tyHermesConfiguration.a_tyDSParam[0].sClientAddress;
			tyCurrentConfigurationSnd.tyData.a_tyDownstreamConfigurations[0].sDownstreamInterfaceId	    := p_tyHermesConfiguration.a_tyDSParam[0].sDownstreamInterfaceId;
			tyCurrentConfigurationSnd.tyData.a_tyDownstreamConfigurations[0].uiPort                 	:= p_tyHermesConfiguration.a_tyDSParam[0].uiSvrPort;

			tyCurrentConfigurationSnd.tyAvl.bMachineId					                              	:= tyCurrentConfigurationSnd.tyData.sMachineId <> '';
			tyCurrentConfigurationSnd.tyAvl.bSupervisorySystemPort		                            	:= tyCurrentConfigurationSnd.tyData.uiSupervisorySystemPort <> 0;
			tyCurrentConfigurationSnd.tyAvl.bUpstreamConfigurations	                            	    := TRUE;
			tyCurrentConfigurationSnd.tyAvl.bDownstreamConfigurations	                            	:= TRUE;
			tyCurrentConfigurationSnd.tyAvl.iUpstreamConfigurations	                                 	:= 1;
			tyCurrentConfigurationSnd.tyAvl.iDownstreamConfigurations	                        	    := 1;
			tyCurrentConfigurationSnd.tyAvl.a_tyUpstreamConfigurations[0].bUpstreamLaneId		        := tyCurrentConfigurationSnd.tyData.a_tyUpstreamConfigurations[0].iUpstreamLaneId <> 0;
			tyCurrentConfigurationSnd.tyAvl.a_tyUpstreamConfigurations[0].bHostAddress		            := tyCurrentConfigurationSnd.tyData.a_tyUpstreamConfigurations[0].sHostAddress <> '';
			tyCurrentConfigurationSnd.tyAvl.a_tyUpstreamConfigurations[0].bUpstreamInterfaceId	        := tyCurrentConfigurationSnd.tyData.a_tyUpstreamConfigurations[0].sUpstreamInterfaceId <> '';
			tyCurrentConfigurationSnd.tyAvl.a_tyUpstreamConfigurations[0].bPort		                    := tyCurrentConfigurationSnd.tyData.a_tyUpstreamConfigurations[0].uiPort <>0;

			tyCurrentConfigurationSnd.tyAvl.a_tyDownstreamConfigurations[0].bDownstreamLaneId	    	:= tyCurrentConfigurationSnd.tyData.a_tyDownstreamConfigurations[0].iDownstreamLaneId <>0;
			tyCurrentConfigurationSnd.tyAvl.a_tyDownstreamConfigurations[0].bClientAddress		        := tyCurrentConfigurationSnd.tyData.a_tyDownstreamConfigurations[0].sClientAddress <> '';
			tyCurrentConfigurationSnd.tyAvl.a_tyDownstreamConfigurations[0].bDownstreamInterfaceId	    := tyCurrentConfigurationSnd.tyData.a_tyDownstreamConfigurations[0].sDownstreamInterfaceId <> '';
			tyCurrentConfigurationSnd.tyAvl.a_tyDownstreamConfigurations[0].bPort		                := tyCurrentConfigurationSnd.tyData.a_tyDownstreamConfigurations[0].uiPort <> 0;

		END_IF

	END_IF

END_ACTION
```

#### Act_Background_SequenceTO.st - Do Not Change!!!
```iecst
(** 2021-08-01 **)
ACTION Act_Background_SequenceTO:

	IF (eStatus1 <> Error) AND (eStatus2 <> Error) THEN

		//Time Out
		fbSequenceTO.eState				:= fbSequenceSvy.eState;
		fbSequenceTO.tConnTimeOut		:= p_tConnTimeOut;
		fbSequenceTO(bEn := TRUE);

		IF fbSequenceTO.udiStatus > 0 AND fbSequenceTO.udiStatus < 65534 THEN

			IF fbSequenceTO.udiStatus = 2912 THEN
				eStatus1	:= Error;
				udiStatus1	:= 10106;	//Supervisory Service Description Interchange Time Out

				fHermesAddOneMsgSend(ADR(a_eMsgSend) , ADR(udiMsgSendBffr) , HermesMsgTypeNotification);

				tyNotificationSnd.tyAvl.bSeverity			:= TRUE;
				tyNotificationSnd.tyAvl.bNotificationCode	:= TRUE;
				tyNotificationSnd.tyAvl.bDescription		:= TRUE;
				tyNotificationSnd.tyData.eSeverity			:= HermesSeverityFatalError;
				tyNotificationSnd.tyData.iNotificationCode	:= UDINT_TO_INT(udiStatus1);
				tyNotificationSnd.tyData.sDescription		:= a_tyAlmText[udiStatus1].sAlmText;

			ELSE
				eStatus2	:= Error;
				udiStatus2	:= fbSequenceTO.udiStatus;

				fHermesAddOneMsgSend(ADR(a_eMsgSend) , ADR(udiMsgSendBffr) , HermesMsgTypeNotification);

				tyNotificationSnd.tyAvl.bSeverity			:= TRUE;
				tyNotificationSnd.tyAvl.bNotificationCode	:= TRUE;
				tyNotificationSnd.tyAvl.bDescription		:= TRUE;
				tyNotificationSnd.tyData.eSeverity			:= HermesSeverityFatalError;
				tyNotificationSnd.tyData.iNotificationCode	:= UDINT_TO_INT(udiStatus2);
				tyNotificationSnd.tyData.sDescription		:= a_tyAlmText[udiStatus2].sAlmText;

			END_IF

		END_IF

	END_IF

END_ACTION
```

#### Act_Background_ChkAlive.st - Do Not Change!!!
```iecst
(** 2021-08-01 **)
ACTION Act_Background_ChkAlive:

	IF eStatus1 <> Error THEN

		//Standard Check Alive (Without Ping & Pong)
		fbCheckAlive.bDataRcv		:= tyMsgTypeRcv.bCheckAlive OR tyMsgTypeRcv.bSetConfiguration OR tyMsgTypeRcv.bGetConfiguration OR tyMsgTypeRcv.bSendWorkOrderInfo;
		fbCheckAlive.tSendTm		:= p_tyParam.tSndAlive;
		fbCheckAlive.tRcvTimeOut	:= p_tyParam.tRcvAlive;
		fbCheckAlive(bEn := TRUE);

		IF fbCheckAlive.udiStatus > 0 AND fbCheckAlive.udiStatus < 65534 THEN
			eStatus1	:= Error;

			IF fbCheckAlive.udiStatus = 2767 THEN
				udiStatus1	:= 10132;	//Check Alive Time Out
			ELSE
				udiStatus1	:= fbCheckAlive.udiStatus;
			END_IF

			fHermesAddOneMsgSend(ADR(a_eMsgSend) , ADR(udiMsgSendBffr) , HermesMsgTypeNotification);

			tyNotificationSnd.tyAvl.bSeverity			:= TRUE;
			tyNotificationSnd.tyAvl.bNotificationCode	:= TRUE;
			tyNotificationSnd.tyAvl.bDescription		:= TRUE;
			tyNotificationSnd.tyData.eSeverity			:= HermesSeverityFatalError;
			tyNotificationSnd.tyData.iNotificationCode	:= UDINT_TO_INT(udiStatus1);
			tyNotificationSnd.tyData.sDescription		:= a_tyAlmText[udiStatus1].sAlmText;

		ELSE
			IF EDGEPOS(fbCheckAlive.bDataSend) THEN
				fHermesAddOneMsgSend(ADR(a_eMsgSend) , ADR(udiMsgSendBffr) , HermesMsgTypeCheckAlive);
				tyCheckAliveSnd	:= fbCheckAlive.tyDataSend;
			END_IF

		END_IF

		tyMsgTypeRcv.bCheckAlive	:= FALSE;	//Reset Check Alive

	END_IF

END_ACTION
```

#### Act_Background_UpdtConfig.st - Do Not Change!!!
```iecst
(** 2021-08-01 **)
ACTION Act_Background_UpdtConfig:

	IF eStatus2 <> Error THEN
		IF tySServiceDescriptionRcv.tyData.tySupportedFeatures.bFeatureConfiguration AND p_tyParam.bFeatureConfiguration THEN

		    IF tyMsgTypeRcv.bSetConfiguration = TRUE THEN

				tySetConfiguration.tyAvl.bMachineId						:= tySetConfigurationRcv.tyAvl.bMachineId;
				tySetConfiguration.tyAvl.bSupervisorySystemPort			:= tySetConfigurationRcv.tyAvl.bSupervisorySystemPort;
				tySetConfiguration.tyAvl.bUpstreamConfigurations		:= tySetConfigurationRcv.tyAvl.bUpstreamConfigurations;
				tySetConfiguration.tyAvl.bDownstreamConfigurations		:= tySetConfigurationRcv.tyAvl.bDownstreamConfigurations;
				tySetConfiguration.tyAvl.iUpstreamConfigurations		:= tySetConfigurationRcv.tyAvl.iUpstreamConfigurations;
				tySetConfiguration.tyAvl.iDownstreamConfigurations		:= tySetConfigurationRcv.tyAvl.iDownstreamConfigurations;
				tySetConfiguration.tyAvl.a_tyUpstreamConfigurations		:= tySetConfigurationRcv.tyAvl.a_tyUpstreamConfigurations;
				tySetConfiguration.tyAvl.a_tyDownstreamConfigurations	:= tySetConfigurationRcv.tyAvl.a_tyDownstreamConfigurations;

				tySetConfiguration.tyData.sMachineId					:= tySetConfigurationRcv.tyData.sMachineId;
				tySetConfiguration.tyData.uiSupervisorySystemPort		:= tySetConfigurationRcv.tyData.uiSupervisorySystemPort;
				tySetConfiguration.tyData.a_tyUpstreamConfigurations	:= tySetConfigurationRcv.tyData.a_tyUpstreamConfigurations;
				tySetConfiguration.tyData.a_tyDownstreamConfigurations	:= tySetConfigurationRcv.tyData.a_tyDownstreamConfigurations;

				udiTargetAddress := ADR(tySetConfiguration.tyData.a_tyUpstreamConfigurations[0].iUpstreamLaneId); //Start address
				udiSizeAddress   := SIZEOF(tySetConfiguration.tyData.a_tyUpstreamConfigurations[0]); //Size of one array

				udiTargetAddress1 := ADR(tySetConfiguration.tyData.a_tyDownstreamConfigurations[0].iDownstreamLaneId); //Start address
				udiSizeAddress1   := SIZEOF(tySetConfiguration.tyData.a_tyDownstreamConfigurations[0]); //Size of one array

				FOR k := 0 TO c_diHermesConfigMaxIdx DO //Max configuration

					IF memcmp((udiTargetAddress)+(k*udiSizeAddress), ADR(j) , 1) = 0 THEN

						bFoundIndexUS1	:= TRUE;
						udiFoundIndexUS1  := k;

						tySetConfigurationModified.tyData.a_tyUpstreamConfigurations[0].iUpstreamLaneId	        := tySetConfiguration.tyData.a_tyUpstreamConfigurations[udiFoundIndexUS1].iUpstreamLaneId;
						tySetConfigurationModified.tyData.a_tyUpstreamConfigurations[0].sHostAddress	        := tySetConfiguration.tyData.a_tyUpstreamConfigurations[udiFoundIndexUS1].sHostAddress;
						tySetConfigurationModified.tyData.a_tyUpstreamConfigurations[0].sUpstreamInterfaceId	:= tySetConfiguration.tyData.a_tyUpstreamConfigurations[udiFoundIndexUS1].sUpstreamInterfaceId;
						tySetConfigurationModified.tyData.a_tyUpstreamConfigurations[0].uiPort              	:= tySetConfiguration.tyData.a_tyUpstreamConfigurations[udiFoundIndexUS1].uiPort;

					ELSIF memcmp((udiTargetAddress)+(k*udiSizeAddress), ADR(jj) , 1) = 0 THEN

						bFoundIndexUS2	:= TRUE;
						udiFoundIndexUS2  := k;

						tySetConfigurationModified.tyData.a_tyUpstreamConfigurations[1].iUpstreamLaneId	        := tySetConfiguration.tyData.a_tyUpstreamConfigurations[udiFoundIndexUS2].iUpstreamLaneId;
						tySetConfigurationModified.tyData.a_tyUpstreamConfigurations[1].sHostAddress	        := tySetConfiguration.tyData.a_tyUpstreamConfigurations[udiFoundIndexUS2].sHostAddress;
						tySetConfigurationModified.tyData.a_tyUpstreamConfigurations[1].sUpstreamInterfaceId	:= tySetConfiguration.tyData.a_tyUpstreamConfigurations[udiFoundIndexUS2].sUpstreamInterfaceId;
						tySetConfigurationModified.tyData.a_tyUpstreamConfigurations[1].uiPort              	:= tySetConfiguration.tyData.a_tyUpstreamConfigurations[udiFoundIndexUS2].uiPort;

					ELSIF memcmp((udiTargetAddress)+(k*udiSizeAddress), ADR(jjj) , 1) = 0 THEN

						bFoundIndexUS3	:= TRUE;
						udiFoundIndexUS3  := k;

						tySetConfigurationModified.tyData.a_tyUpstreamConfigurations[2].iUpstreamLaneId	        := tySetConfiguration.tyData.a_tyUpstreamConfigurations[udiFoundIndexUS3].iUpstreamLaneId;
						tySetConfigurationModified.tyData.a_tyUpstreamConfigurations[2].sHostAddress	        := tySetConfiguration.tyData.a_tyUpstreamConfigurations[udiFoundIndexUS3].sHostAddress;
						tySetConfigurationModified.tyData.a_tyUpstreamConfigurations[2].sUpstreamInterfaceId	:= tySetConfiguration.tyData.a_tyUpstreamConfigurations[udiFoundIndexUS3].sUpstreamInterfaceId;
						tySetConfigurationModified.tyData.a_tyUpstreamConfigurations[2].uiPort              	:= tySetConfiguration.tyData.a_tyUpstreamConfigurations[udiFoundIndexUS3].uiPort;

					ELSIF memcmp((udiTargetAddress)+(k*udiSizeAddress), ADR(jjjj) , 1) = 0 THEN

						bFoundIndexUS4	:= TRUE;
						udiFoundIndexUS4  := k;

						tySetConfigurationModified.tyData.a_tyUpstreamConfigurations[3].iUpstreamLaneId	        := tySetConfiguration.tyData.a_tyUpstreamConfigurations[udiFoundIndexUS3].iUpstreamLaneId;
						tySetConfigurationModified.tyData.a_tyUpstreamConfigurations[3].sHostAddress	        := tySetConfiguration.tyData.a_tyUpstreamConfigurations[udiFoundIndexUS3].sHostAddress;
						tySetConfigurationModified.tyData.a_tyUpstreamConfigurations[3].sUpstreamInterfaceId	:= tySetConfiguration.tyData.a_tyUpstreamConfigurations[udiFoundIndexUS3].sUpstreamInterfaceId;
						tySetConfigurationModified.tyData.a_tyUpstreamConfigurations[3].uiPort              	:= tySetConfiguration.tyData.a_tyUpstreamConfigurations[udiFoundIndexUS3].uiPort;

					END_IF

				END_FOR

				FOR kk := 0 TO c_diHermesConfigMaxIdx DO //Max configuration

					IF memcmp((udiTargetAddress1)+(kk*udiSizeAddress1), ADR(j) , 1) = 0 THEN

						bFoundIndexDS1	:= TRUE;
						udiFoundIndexDS1  := kk;

						tySetConfigurationModified.tyData.a_tyDownstreamConfigurations[0].iDownstreamLaneId	        := tySetConfiguration.tyData.a_tyDownstreamConfigurations[udiFoundIndexDS1].iDownstreamLaneId;
						tySetConfigurationModified.tyData.a_tyDownstreamConfigurations[0].sClientAddress	        := tySetConfiguration.tyData.a_tyDownstreamConfigurations[udiFoundIndexDS1].sClientAddress;
						tySetConfigurationModified.tyData.a_tyDownstreamConfigurations[0].sDownstreamInterfaceId	:= tySetConfiguration.tyData.a_tyDownstreamConfigurations[udiFoundIndexDS1].sDownstreamInterfaceId;
						tySetConfigurationModified.tyData.a_tyDownstreamConfigurations[0].uiPort                 	:= tySetConfiguration.tyData.a_tyDownstreamConfigurations[udiFoundIndexDS1].uiPort;

					ELSIF memcmp((udiTargetAddress1)+(kk*udiSizeAddress1), ADR(jj) , 1) = 0 THEN

						bFoundIndexDS2	:= TRUE;
						udiFoundIndexDS2  := kk;

						tySetConfigurationModified.tyData.a_tyDownstreamConfigurations[1].iDownstreamLaneId	        := tySetConfiguration.tyData.a_tyDownstreamConfigurations[udiFoundIndexDS2].iDownstreamLaneId;
						tySetConfigurationModified.tyData.a_tyDownstreamConfigurations[1].sClientAddress	        := tySetConfiguration.tyData.a_tyDownstreamConfigurations[udiFoundIndexDS2].sClientAddress;
						tySetConfigurationModified.tyData.a_tyDownstreamConfigurations[1].sDownstreamInterfaceId	:= tySetConfiguration.tyData.a_tyDownstreamConfigurations[udiFoundIndexDS2].sDownstreamInterfaceId;
						tySetConfigurationModified.tyData.a_tyDownstreamConfigurations[1].uiPort                 	:= tySetConfiguration.tyData.a_tyDownstreamConfigurations[udiFoundIndexDS2].uiPort;

					ELSIF memcmp((udiTargetAddress1)+(kk*udiSizeAddress1), ADR(jjj) , 1) = 0 THEN

						bFoundIndexDS3	:= TRUE;
						udiFoundIndexDS3  := kk;

						tySetConfigurationModified.tyData.a_tyDownstreamConfigurations[2].iDownstreamLaneId	        := tySetConfiguration.tyData.a_tyDownstreamConfigurations[udiFoundIndexDS3].iDownstreamLaneId;
						tySetConfigurationModified.tyData.a_tyDownstreamConfigurations[2].sClientAddress	        := tySetConfiguration.tyData.a_tyDownstreamConfigurations[udiFoundIndexDS3].sClientAddress;
						tySetConfigurationModified.tyData.a_tyDownstreamConfigurations[2].sDownstreamInterfaceId	:= tySetConfiguration.tyData.a_tyDownstreamConfigurations[udiFoundIndexDS3].sDownstreamInterfaceId;
						tySetConfigurationModified.tyData.a_tyDownstreamConfigurations[2].uiPort                 	:= tySetConfiguration.tyData.a_tyDownstreamConfigurations[udiFoundIndexDS3].uiPort;

					ELSIF memcmp((udiTargetAddress1)+(kk*udiSizeAddress1), ADR(jjjj) , 1) = 0 THEN

						bFoundIndexDS4	:= TRUE;
						udiFoundIndexDS4  := kk;

						tySetConfigurationModified.tyData.a_tyDownstreamConfigurations[3].iDownstreamLaneId	        := tySetConfiguration.tyData.a_tyDownstreamConfigurations[udiFoundIndexDS4].iDownstreamLaneId;
						tySetConfigurationModified.tyData.a_tyDownstreamConfigurations[3].sClientAddress	        := tySetConfiguration.tyData.a_tyDownstreamConfigurations[udiFoundIndexDS4].sClientAddress;
						tySetConfigurationModified.tyData.a_tyDownstreamConfigurations[3].sDownstreamInterfaceId	:= tySetConfiguration.tyData.a_tyDownstreamConfigurations[udiFoundIndexDS4].sDownstreamInterfaceId;
						tySetConfigurationModified.tyData.a_tyDownstreamConfigurations[3].uiPort                 	:= tySetConfiguration.tyData.a_tyDownstreamConfigurations[udiFoundIndexDS4].uiPort;
					END_IF

				END_FOR

				tySetConfigurationModified.tyAvl.bMachineId				        := tySetConfiguration.tyAvl.bMachineId;
				tySetConfigurationModified.tyAvl.bSupervisorySystemPort			:= tySetConfiguration.tyAvl.bSupervisorySystemPort;
				tySetConfigurationModified.tyAvl.bUpstreamConfigurations		:= tySetConfiguration.tyAvl.bUpstreamConfigurations;
				tySetConfigurationModified.tyAvl.bDownstreamConfigurations		:= tySetConfiguration.tyAvl.bDownstreamConfigurations;
				tySetConfigurationModified.tyAvl.iUpstreamConfigurations		:= tySetConfiguration.tyAvl.iUpstreamConfigurations;
				tySetConfigurationModified.tyAvl.iDownstreamConfigurations		:= tySetConfiguration.tyAvl.iDownstreamConfigurations;
				tySetConfigurationModified.tyAvl.a_tyUpstreamConfigurations		:= tySetConfiguration.tyAvl.a_tyUpstreamConfigurations;
				tySetConfigurationModified.tyAvl.a_tyDownstreamConfigurations	:= tySetConfiguration.tyAvl.a_tyDownstreamConfigurations;

				tySetConfigurationModified.tyData.sMachineId					:= tySetConfiguration.tyData.sMachineId;
				tySetConfigurationModified.tyData.uiSupervisorySystemPort		:= tySetConfiguration.tyData.uiSupervisorySystemPort;

				IF bUpdateUIData = FALSE THEN
					bWriteConfig := TRUE;
					tyMsgTypeRcv.bSetConfiguration	:= FALSE;
				END_IF

			END_IF
		ELSE

			bWriteConfig := FALSE;
			tyMsgTypeRcv.bSetConfiguration := FALSE;
		END_IF

	END_IF

END_ACTION
```

#### Act_Background_ChgConfig.st - Do Not Change!!!
```iecst
(** 2021-08-01 **)
ACTION Act_Background_ChgConfig:

	IF eStatus2 <> Error THEN

		IF (tyParamOld.uiSvySvstemPort <> p_tyParam.uiSvySvstemPort)
			OR (tyParamOld.bFeatureBoardTracking <> p_tyParam.bFeatureBoardTracking) OR (tyParamOld.bFeatureCheckAliveResponse <> p_tyParam.bFeatureCheckAliveResponse) OR (tyParamOld.bFeatureConfiguration <> p_tyParam.bFeatureConfiguration)
			OR (tyParamOld.bFeatureQueryWorkOrderInfo <> p_tyParam.bFeatureQueryWorkOrderInfo) (*OR (tyParamOld.bFeatureSendWorkOrderInfo <> p_tyParam.bFeatureSendWorkOrderInfo)*) THEN

			IF udiClntIdent <> 0 THEN
				fHermesAddOneMsgSend(ADR(a_eMsgSend) , ADR(udiMsgSendBffr) , HermesMsgTypeNotification);

				tyNotificationSnd.tyAvl.bSeverity			:= TRUE;
				tyNotificationSnd.tyAvl.bNotificationCode	:= TRUE;
				tyNotificationSnd.tyAvl.bDescription		:= TRUE;
				tyNotificationSnd.tyData.eSeverity			:= HermesSeverityFatalError;
				tyNotificationSnd.tyData.iNotificationCode	:= 3;
				tyNotificationSnd.tyData.sDescription		:= 'Configuration Changed';

			END_IF

			bRstConnection	:= TRUE;

		END_IF

	END_IF

END_ACTION
```

#### Act_Background_NotificationSnd.st - Do Not Change!!!
```iecst
(** 2021-08-01 **)
ACTION Act_Background_NotificationSnd:

	IF a_eMsgSend[0] = HermesMsgTypeNotification THEN
		bRstConnection	:= fHermesNotificationRstConn(tyNotificationSnd) OR bRstConnection;
//		bRstState		:= fHermesNotificationRstState(tyNotificationSnd) OR bRstState;
	END_IF

END_ACTION
```

#### Act_Background_QueryWorkOrderInfo.st - Do Not Change!!!
```iecst
(** 2021-08-01 **)
ACTION Act_Background_QueryWorkOrderInfo:

	IF eStatus2 <> Error THEN

		IF EDGEPOS(p_bQueryWorkOrderInfo OR p_bReinsertBrd) AND p_bAcceptCondition THEN //Hermes 1.3 Board Reinsert Function

			fHermesAddOneMsgSend(ADR(a_eMsgSend) , ADR(udiMsgSendBffr) , HermesMsgTypeQueryWorkOrderInfo);

			fHermesGenerateUUID(ADR(tyQueryWorkOrderInfo.tyData.sQueryId) , p_tyDTStructure , pa_usiMacAddr); //Generate QueryID

			tyQueryWorkOrderInfo.tyData.sMachineId							:= p_sMcId;
			tyQueryWorkOrderInfo.tyData.sMagazineId							:= p_sMagazineId;
			tyQueryWorkOrderInfo.tyData.iSlotId								:= p_iSlotId;
			tyQueryWorkOrderInfo.tyData.sBarcode						    := p_sBarcode;

			tyQueryWorkOrderInfo.tyAvl.bQueryId							    := tyQueryWorkOrderInfo.tyData.sQueryId <> '';
			tyQueryWorkOrderInfo.tyAvl.bMachineId							:= tyQueryWorkOrderInfo.tyData.sMachineId <> '';
			tyQueryWorkOrderInfo.tyAvl.bMagazineId							:= tyQueryWorkOrderInfo.tyData.sMagazineId <> '';
			tyQueryWorkOrderInfo.tyAvl.bSlotId								:= tyQueryWorkOrderInfo.tyData.iSlotId <> 0;
			tyQueryWorkOrderInfo.tyAvl.bBarcode								:= tyQueryWorkOrderInfo.tyData.sBarcode <> '';
			bQueryInsertBoard   	:= TRUE;	//Hermes 1.3 Board Reinsert Function
			bRcvInsertBoardInfo		:= FALSE;	//Hermes 1.3 Board Reinsert Function
			bManualInsertData       := FALSE;	//Hermes 1.3 Board Reinsert Function
			bReplyWorkOrderInfo     := FALSE;
			bRcvWorkOrderInfo2      := FALSE;
		END_IF

		IF (p_bQueryWorkOrderInfo OR p_bReinsertBrd) AND p_bAcceptCondition = FALSE THEN
			bRstWorkOrderInfo := TRUE;
		END_IF

		IF tyMsgTypeRcv.bSendWorkOrderInfo THEN

			IF (p_bQueryWorkOrderInfo OR p_bReinsertBrd) AND (udiStatus2 = 0) THEN //After CmpParamRcv
				IF tySendWorkOrderInfoRcv.tyAvl.bWorkOrderId AND tySendWorkOrderInfoRcv.tyData.sWorkOrderId <> '' AND p_bAcceptCondition AND
					tySendWorkOrderInfoRcv.tyData.rWidth >= 50.0 AND tySendWorkOrderInfoRcv.tyData.rWidth <= 460.0 THEN //Wait Accept Conditon On

					//bRcvWorkOrderInfo1 := TRUE;
					bRcvWorkOrderInfo2  := FALSE;
					bRcvInsertBoardInfo := TRUE;
					tySendWorkOrderInfoAcc := tySendWorkOrderInfoRcv;
					tyMsgTypeRcv.bSendWorkOrderInfo := FALSE;
					sWorkOrderId := tySendWorkOrderInfoAcc.tyData.sWorkOrderId;

				ELSIF (tySendWorkOrderInfoRcv.tyAvl.bWorkOrderId = FALSE OR tySendWorkOrderInfoRcv.tyData.sWorkOrderId = '') OR
					tySendWorkOrderInfoRcv.tyData.rWidth < 50.0 OR tySendWorkOrderInfoRcv.tyData.rWidth > 460.0THEN
					bRcvWorkOrderInfo2 := TRUE;
					bRcvInsertBoardInfo := FALSE;
					tyMsgTypeRcv.bSendWorkOrderInfo := FALSE;
				END_IF

			ELSIF (p_bQueryWorkOrderInfo = FALSE OR p_bReinsertBrd = FALSE) THEN
				tyMsgTypeRcv.bSendWorkOrderInfo := FALSE;
			END_IF

		END_IF

		IF 	bRcvWorkOrderInfo1 = TRUE AND NOT(p_bHermesSvyQueryBoardInfo OR p_bReinsertBrd) THEN

			tyInfoData1.sProgNm		:= p_sProgNm;
			tyInfoData1.udiCode		:= 10000;
			tyInfoData1.eSeverity	:= AlmSeverityInfo;
			tyInfoData1.sAlmMsg		:= p_sInfoMsg1;

		ELSIF bRcvWorkOrderInfo2 = TRUE THEN

			tyInfoData2.sProgNm		:= p_sProgNm;
			tyInfoData2.udiCode		:= 10000;
			tyInfoData2.eSeverity	:= AlmSeverityInfo;
			tyInfoData2.sAlmMsg		:= p_sInfoMsg2;

		END_IF

		IF  bRstWorkOrderInfo = TRUE THEN

			tyInfoData3.sProgNm		:= p_sProgNm;
			tyInfoData3.udiCode		:= 10000;
			tyInfoData3.eSeverity	:= AlmSeverityInfo;
			tyInfoData3.sAlmMsg		:= p_sInfoMsg3;

		END_IF

		IF 	EDGEPOS(bQueryInsertBoard) THEN

			tyInfoData4.sProgNm		:= p_sProgNm;
			tyInfoData4.udiCode		:= 10000;
			tyInfoData4.eSeverity	:= AlmSeverityInfo;
			tyInfoData4.sAlmMsg		:= p_sInfoMsg4;

		ELSIF EDGEPOS(p_bAcceptCondition = TRUE AND bManualInsertData AND p_bAWWidthPosDiff = FALSE) THEN
			tyInfoData4.sProgNm		:= '';                   //Clear previous message
			tyInfoData4.udiCode		:= 0;
			tyInfoData4.eSeverity	:= AlmSeverityNA;
			tyInfoData4.sAlmMsg		:= '';

			tyInfoData5.sProgNm		:= p_sProgNm;
			tyInfoData5.udiCode		:= 10000;
			tyInfoData5.eSeverity	:= AlmSeverityInfo;
			tyInfoData5.sAlmMsg		:= p_sInfoMsg5;
			                                                                                                                                                                                                                                                                                       //Debug
		ELSIF (EDGEPOS (bQueryInsertBoard AND (p_bConvRgtSen OR p_bConvLftSen)) OR EDGEPOS(bRcvInsertBoardInfo= FALSE AND p_eLinkMcParamDSCommMod = McSetCommModHermes AND p_tyMcParamCurr.bHermesSvyEn AND p_tyNtParamCurr.bHermesBrdReInsertPrep AND (p_bConvRgtSen OR p_bConvLftSen)) OR EDGEPOS(bManualInsertData AND p_bConvLftSen))  AND NOT p_bOpsGConvStepDSTmr AND NOT p_bOpsGConvStepDSCommTmr AND NOT p_bOpsGConvStepEntBrd AND p_bOpsRun THEN
			tyInfoData6.sProgNm		:= p_sProgNm;
			tyInfoData6.udiCode		:= 10000;
			tyInfoData6.eSeverity	:= AlmSeverityInfo;
			tyInfoData6.sAlmMsg		:= p_sInfoMsg6;

		END_IF

		IF EDGEPOS(bRcvInsertBoardInfo OR bRcvWorkOrderInfo2) AND udiStatus2 = 0 THEN
			fHermesAddOneMsgSend(ADR(a_eMsgSend) , ADR(udiMsgSendBffr) , HermesMsgTypeReplyWorkOrderInfo);

			IF  bRcvInsertBoardInfo AND p_bAcceptCondition  THEN
				tyReplyWorkOrderInfo.tyData.sWorkOrderId					    := tySendWorkOrderInfoAcc.tyData.sWorkOrderId;
				tyReplyWorkOrderInfo.tyData.sBatchId					      	:= tySendWorkOrderInfoAcc.tyData.sBatchId;
				tyReplyWorkOrderInfo.tyData.iStatus							    := 1;          //WorkOrder accepted
				bReplyWorkOrderInfo                                             := TRUE;
			ELSIF bRcvWorkOrderInfo2 THEN
				tyReplyWorkOrderInfo.tyData.sWorkOrderId					    := tySendWorkOrderInfoRcv.tyData.sWorkOrderId;
				tyReplyWorkOrderInfo.tyData.sBatchId					      	:= tySendWorkOrderInfoRcv.tyData.sBatchId;
				tyReplyWorkOrderInfo.tyData.iStatus							    := 0;         //WorkOrder Rejected
				bRcvWorkOrderInfo2                                              := FALSE;
			ELSE
				tyReplyWorkOrderInfo.tyData.sWorkOrderId					    := tySendWorkOrderInfoAcc.tyData.sWorkOrderId;
				tyReplyWorkOrderInfo.tyData.sBatchId					      	:= tySendWorkOrderInfoAcc.tyData.sBatchId;
				tyReplyWorkOrderInfo.tyData.iStatus							    := 2;          //WorkOrder accepted and queue
				bReplyWorkOrderInfo                                             := TRUE;
			END_IF

			tyReplyWorkOrderInfo.tyAvl.bWorkOrderId					:= tyReplyWorkOrderInfo.tyData.sWorkOrderId <> '';
			tyReplyWorkOrderInfo.tyAvl.bBatchId                     := tyReplyWorkOrderInfo.tyData.sBatchId <> '';
			tyReplyWorkOrderInfo.tyAvl.bStatus                      :=  TRUE;
		END_IF

		//Hermes 1.3 Board Reinsert Function
		IF (p_bQueryWorkOrderInfo OR p_bReinsertBrd) AND p_bAcceptCondition AND tySendWorkOrderInfoRcv.tyAvl.bWidth AND bRcvInsertBoardInfo THEN                  // ADD for 2023-0061E01SSJob
			//tySendWorkOrderInfoNewRcv := tySendWorkOrderInfoRcv;
			diReqWidthInUM := REAL_TO_DINT(tySendWorkOrderInfoRcv.tyData.rWidth*1000);
			sWorkOrderId := tySendWorkOrderInfoRcv.tyData.sWorkOrderId;
			sBatchId := tySendWorkOrderInfoRcv.tyData.sBatchId;
			//sRecipeNm	:= tySendWorkOrderInfoRcv.tyData.sProductTypeId;	//Add On
			p_tyProdRcpCurrRcp.diWidthInUM	:= diReqWidthInUM;
			bQueryInsertBoard   := FALSE;
			//bRcvInsertBoardInfo := FALSE;
			bManualInsertData := TRUE;
			tySendWorkOrderInfoRcv.tyAvl.bWidth:= FALSE;
		END_IF

		IF ((p_bQueryWorkOrderInfo = FALSE AND bQueryInsertBoard = FALSE) AND NOT(p_bConvRgtSen)) THEN	//Hermes 1.3 Board Reinsert Function

			//Clear Info Message 1
			tyInfoData1.sProgNm		:= '';
			tyInfoData1.udiCode		:= 0;
			tyInfoData1.eSeverity	:= AlmSeverityNA;
			tyInfoData1.sAlmMsg		:= '';
			bRcvWorkOrderInfo1 := FALSE;

			//Clear Info Message 2
			tyInfoData2.sProgNm		:= '';
			tyInfoData2.udiCode		:= 0;
			tyInfoData2.eSeverity	:= AlmSeverityNA;
			tyInfoData2.sAlmMsg		:= '';
			bRcvWorkOrderInfo2 := FALSE;

			//Clear Info Message 3
			tyInfoData3.sProgNm		:= '';
			tyInfoData3.udiCode		:= 0;
			tyInfoData3.eSeverity	:= AlmSeverityNA;
			tyInfoData3.sAlmMsg		:= '';
			bRstWorkOrderInfo := FALSE;

			//Clear Info Message 4
			tyInfoData4.sProgNm		:= '';
			tyInfoData4.udiCode		:= 0;
			tyInfoData4.eSeverity	:= AlmSeverityNA;
			tyInfoData4.sAlmMsg		:= '';

		ELSIF (p_bReinsertBrd = FALSE AND p_bConvRgtSen) THEN
			//Clear Info Message 5
			tyInfoData5.sProgNm		:= '';
			tyInfoData5.udiCode		:= 0;
			tyInfoData5.eSeverity	:= AlmSeverityNA;
			tyInfoData5.sAlmMsg		:= '';
			bQueryInsertBoard   	:= FALSE;
			//bRcvInsertBoardInfo		:= FALSE;
		ELSIF EDGENEG(p_bConvRgtSen) AND (p_bHermesSvyQueryBoardInfo OR p_bHermesReinsertBoard) THEN
			bRcvWorkOrderInfo1 := FALSE;
		END_IF

		IF (EDGENEG (p_bConvRgtSen OR p_bConvLftSen)) AND  tyInfoData6.udiCode <> 0  THEN
			//Clear Info Message 6
			tyInfoData6.sProgNm		:= '';
			tyInfoData6.udiCode		:= 0;
			tyInfoData6.eSeverity	:= AlmSeverityNA;
			tyInfoData6.sAlmMsg		:= '';
		END_IF

		//Hermes 1.3 Board Reinsert Function		//Distrigger Insert Brd Btn
		IF EDGENEG (p_bConvRgtSen) OR NOT p_bOpsRun OR (EDGENEG(p_bInsertBoard) AND NOT(p_bConvRgtSen)) THEN
			bRcvInsertBoardInfo		:= FALSE;
			bManualInsertData       := FALSE;
			tyInfoData5.sProgNm		:= '';
			tyInfoData5.udiCode		:= 0;
			tyInfoData5.eSeverity	:= AlmSeverityNA;
			tyInfoData5.sAlmMsg		:= '';
			bQueryInsertBoard   	:= FALSE;

		END_IF

		//Hermes 1.3 Board Reinsert Function
		IF p_bInsertBoard= FALSE THEN
			bQueryInsertBoard := FALSE;
		END_IF

	END_IF

	IF p_bOpsRun = FALSE OR eStatus2 = Error (*OR eStatus1 = Error OR eStatus3 = Error*) THEN	//Debug
		//Clear Info Message 5
		tyInfoData5.sProgNm		:= '';
		tyInfoData5.udiCode		:= 0;
		tyInfoData5.eSeverity	:= AlmSeverityNA;
		tyInfoData5.sAlmMsg		:= '';
		bQueryInsertBoard   	:= FALSE;

		tyInfoData4.sProgNm		:= '';
		tyInfoData4.udiCode		:= 0;
		tyInfoData4.eSeverity	:= AlmSeverityNA;
		tyInfoData4.sAlmMsg		:= '';
		tySendWorkOrderInfoRcv.tyAvl.bWidth := FALSE;
	END_IF

END_ACTION
```

#### Act_Background_SendBoardArrivedLane1.st - Do Not Change!!!
```iecst
(** 2021-08-01 **)
ACTION Act_Background_SendBoardArrivedLane1: //Send after our machine send out "StopTransport" message to upstream

	IF eStatus2 <> Error THEN
		IF tySServiceDescriptionRcv.tyData.tySupportedFeatures.bFeatureBoardTracking = TRUE AND p_tyParam.bFeatureBoardTracking AND bHandshakeDone THEN
			IF EDGEPOS(p_bUSHermesStopTransport1) THEN

				fHermesAddOneMsgSend(ADR(a_eMsgSend) , ADR(udiMsgSendBffr) , HermesMsgTypeBoardArrived1);

				tyBoardArrived1.tyData.sMachineId     	        := p_sMcId;
				tyBoardArrived1.tyData.iUpstreamLaneId    	    := p_tyHermesConfiguration.a_tyUSParam[0].iLaneID;
				tyBoardArrived1.tyData.sUpstreamInterfaceId     := p_tyHermesConfiguration.a_tyUSParam[0].sUpstreamInterfaceId;
				tyBoardArrived1.tyData.sMagazineId           	:= sMagazineId;
				tyBoardArrived1.tyData.iSlotId     	            := iSlotId;
				tyBoardArrived1.tyData.eBoadTransfer    	    := HermesTransferred;
				tyBoardArrived1.tyData.sBoardId     	        := p_tyUSBoardArrived1.tyData.sBoardId;
				tyBoardArrived1.tyData.sBoardIdCreatedBy     	:= p_tyUSBoardArrived1.tyData.sBoardIdCreatedBy;
				tyBoardArrived1.tyData.eFailedBoard				:= p_tyUSBoardArrived1.tyData.eFailedBoard;
				tyBoardArrived1.tyData.sProductTypeId			:= p_tyUSBoardArrived1.tyData.sProductTypeId;
				tyBoardArrived1.tyData.eFlippedBoard		  	:= p_tyUSBoardArrived1.tyData.eFlippedBoard;
				tyBoardArrived1.tyData.sTopBarcode				:= p_tyUSBoardArrived1.tyData.sTopBarcode;
				tyBoardArrived1.tyData.sBottomBarcode			:= p_tyUSBoardArrived1.tyData.sBottomBarcode;
				tyBoardArrived1.tyData.rLength					:= p_tyUSBoardArrived1.tyData.rLength;
				tyBoardArrived1.tyData.rWidth				    := p_tyUSBoardArrived1.tyData.rWidth;
				tyBoardArrived1.tyData.rThickness				:= p_tyUSBoardArrived1.tyData.rThickness;
				tyBoardArrived1.tyData.rConveyorSpeed		    := p_tyUSBoardArrived1.tyData.rConveyorSpeed;
				tyBoardArrived1.tyData.rTopClearanceHeight		:= p_tyUSBoardArrived1.tyData.rTopClearanceHeight;
				tyBoardArrived1.tyData.rBottomClearanceHeight	:= p_tyUSBoardArrived1.tyData.rBottomClearanceHeight;
				tyBoardArrived1.tyData.rWeight					:= p_tyUSBoardArrived1.tyData.rWeight;
				tyBoardArrived1.tyData.sWorkOrdedId             := p_tyUSBoardArrived1.tyData.sWorkOrderId;
				tyBoardArrived1.tyData.sBatchId                 := p_tyUSBoardArrived1.tyData.sBatchId;

			    tyBoardArrived1.tyAvl.bMachineId				:= tyBoardArrived1.tyData.sMachineId <> '';
		     	tyBoardArrived1.tyAvl.bUpstreamLaneId			:= tyBoardArrived1.tyData.iUpstreamLaneId <> 0;
		    	tyBoardArrived1.tyAvl.bUpstreamInterfaceId		:= tyBoardArrived1.tyData.sUpstreamInterfaceId <> '';
		    	tyBoardArrived1.tyAvl.bMagazineId		    	:= tyBoardArrived1.tyData.sMagazineId <> '';
		    	tyBoardArrived1.tyAvl.bSlotId				    := tyBoardArrived1.tyData.iSlotId <> 0;
		    	tyBoardArrived1.tyAvl.bBoardTransfer			:= TRUE;
				tyBoardArrived1.tyAvl.bBoardId					:= tyBoardArrived1.tyData.sBoardId <> '';
				tyBoardArrived1.tyAvl.bBoardIdCreatedBy			:= tyBoardArrived1.tyData.sBoardIdCreatedBy <> '';
				tyBoardArrived1.tyAvl.bFailedBoard				:= TRUE;
				tyBoardArrived1.tyAvl.bProductTypeId		  	:= tyBoardArrived1.tyData.sProductTypeId <> '';
				tyBoardArrived1.tyAvl.bFlippedBoard				:= TRUE;
				tyBoardArrived1.tyAvl.bTopBarcode			    := tyBoardArrived1.tyData.sTopBarcode <> '';
				tyBoardArrived1.tyAvl.bBottomBarcode		   	:= tyBoardArrived1.tyData.sBottomBarcode <> '';
				tyBoardArrived1.tyAvl.bLength				    := tyBoardArrived1.tyData.rLength <> 0;
				tyBoardArrived1.tyAvl.bWidth				  	:= (tyBoardArrived1.tyData.rWidth <> 0);
				tyBoardArrived1.tyAvl.bThickness			   	:= (tyBoardArrived1.tyData.rThickness <> 0);
				tyBoardArrived1.tyAvl.bConveyorSpeed		   	:= tyBoardArrived1.tyData.rConveyorSpeed <> 0;
				tyBoardArrived1.tyAvl.bTopClearanceHeight	    := (tyBoardArrived1.tyData.rTopClearanceHeight <> 0);
				tyBoardArrived1.tyAvl.bBottomClearanceHeight    := (tyBoardArrived1.tyData.rBottomClearanceHeight <> 0);
		    	tyBoardArrived1.tyAvl.bWeight				    := tyBoardArrived1.tyData.rWeight <> 0;
				tyBoardArrived1.tyAvl.bWorkOrderId				:= tyBoardArrived1.tyData.sWorkOrdedId <> '';
				tyBoardArrived1.tyAvl.bBatchId			    	:= tyBoardArrived1.tyData.sBatchId <> '';

			END_IF

		END_IF

	END_IF

END_ACTION
```

#### Act_Background_SendBoardArrivedLane2.st - Do Not Change!!!
```iecst
(** 2021-08-01 **)
ACTION Act_Background_SendBoardArrivedLane2: //Send after our machine send out "StopTransport" message to upstream

	IF eStatus2 <> Error THEN
		IF tySServiceDescriptionRcv.tyData.tySupportedFeatures.bFeatureBoardTracking = TRUE AND p_tyParam.bFeatureBoardTracking AND bHandshakeDone THEN
			IF EDGEPOS(p_bUSHermesStopTransport2) THEN

				fHermesAddOneMsgSend(ADR(a_eMsgSend) , ADR(udiMsgSendBffr) , HermesMsgTypeBoardArrived2);

				tyBoardArrived2.tyData.sMachineId     	        := p_sMcId;
				tyBoardArrived2.tyData.iUpstreamLaneId    	    := p_tyHermesConfiguration.a_tyUSParam[1].iLaneID;
				tyBoardArrived2.tyData.sUpstreamInterfaceId     := p_tyHermesConfiguration.a_tyUSParam[1].sUpstreamInterfaceId;
				tyBoardArrived2.tyData.sMagazineId           	:= sMagazineId;
				tyBoardArrived2.tyData.iSlotId     	            := iSlotId;
				tyBoardArrived2.tyData.eBoadTransfer    	    := HermesTransferred;
				tyBoardArrived2.tyData.sBoardId     	        := p_tyUSBoardArrived2.tyData.sBoardId;
				tyBoardArrived2.tyData.sBoardIdCreatedBy     	:= p_tyUSBoardArrived2.tyData.sBoardIdCreatedBy;
				tyBoardArrived2.tyData.eFailedBoard				:= p_tyUSBoardArrived2.tyData.eFailedBoard;
				tyBoardArrived2.tyData.sProductTypeId			:= p_tyUSBoardArrived2.tyData.sProductTypeId;
				tyBoardArrived2.tyData.eFlippedBoard		  	:= p_tyUSBoardArrived2.tyData.eFlippedBoard;
				tyBoardArrived2.tyData.sTopBarcode				:= p_tyUSBoardArrived2.tyData.sTopBarcode;
				tyBoardArrived2.tyData.sBottomBarcode			:= p_tyUSBoardArrived2.tyData.sBottomBarcode;
				tyBoardArrived2.tyData.rLength					:= p_tyUSBoardArrived2.tyData.rLength;
				tyBoardArrived2.tyData.rWidth				    := p_tyUSBoardArrived2.tyData.rWidth;
				tyBoardArrived2.tyData.rThickness				:= p_tyUSBoardArrived2.tyData.rThickness;
				tyBoardArrived2.tyData.rConveyorSpeed		    := p_tyUSBoardArrived2.tyData.rConveyorSpeed;
				tyBoardArrived2.tyData.rTopClearanceHeight		:= p_tyUSBoardArrived2.tyData.rTopClearanceHeight;
				tyBoardArrived2.tyData.rBottomClearanceHeight	:= p_tyUSBoardArrived2.tyData.rBottomClearanceHeight;
				tyBoardArrived2.tyData.rWeight					:= p_tyUSBoardArrived2.tyData.rWeight;
				tyBoardArrived2.tyData.sWorkOrdedId             := p_tyUSBoardArrived2.tyData.sWorkOrderId;
				tyBoardArrived2.tyData.sBatchId                 := p_tyUSBoardArrived2.tyData.sBatchId;

			    tyBoardArrived2.tyAvl.bMachineId				:= tyBoardArrived2.tyData.sMachineId <> '';
		     	tyBoardArrived2.tyAvl.bUpstreamLaneId			:= tyBoardArrived2.tyData.iUpstreamLaneId <> 0;
		    	tyBoardArrived2.tyAvl.bUpstreamInterfaceId		:= tyBoardArrived2.tyData.sUpstreamInterfaceId <> '';
		    	tyBoardArrived2.tyAvl.bMagazineId		    	:= tyBoardArrived2.tyData.sMagazineId <> '';
		    	tyBoardArrived2.tyAvl.bSlotId				    := tyBoardArrived2.tyData.iSlotId <> 0;
		    	tyBoardArrived2.tyAvl.bBoardTransfer			:= TRUE;
				tyBoardArrived2.tyAvl.bBoardId					:= tyBoardArrived2.tyData.sBoardId <> '';
				tyBoardArrived2.tyAvl.bBoardIdCreatedBy			:= tyBoardArrived2.tyData.sBoardIdCreatedBy <> '';
				tyBoardArrived2.tyAvl.bFailedBoard				:= TRUE;
				tyBoardArrived2.tyAvl.bProductTypeId		  	:= tyBoardArrived2.tyData.sProductTypeId <> '';
				tyBoardArrived2.tyAvl.bFlippedBoard				:= TRUE;
				tyBoardArrived2.tyAvl.bTopBarcode			    := tyBoardArrived2.tyData.sTopBarcode <> '';
				tyBoardArrived2.tyAvl.bBottomBarcode		   	:= tyBoardArrived2.tyData.sBottomBarcode <> '';
				tyBoardArrived2.tyAvl.bLength				    := tyBoardArrived2.tyData.rLength <> 0;
				tyBoardArrived2.tyAvl.bWidth				  	:= (tyBoardArrived2.tyData.rWidth <> 0);
				tyBoardArrived2.tyAvl.bThickness			   	:= (tyBoardArrived2.tyData.rThickness <> 0);
				tyBoardArrived2.tyAvl.bConveyorSpeed		   	:= tyBoardArrived2.tyData.rConveyorSpeed <> 0;
				tyBoardArrived2.tyAvl.bTopClearanceHeight	    := (tyBoardArrived2.tyData.rTopClearanceHeight <> 0);
				tyBoardArrived2.tyAvl.bBottomClearanceHeight    := (tyBoardArrived2.tyData.rBottomClearanceHeight <> 0);
		    	tyBoardArrived2.tyAvl.bWeight				    := tyBoardArrived2.tyData.rWeight <> 0;
				tyBoardArrived2.tyAvl.bWorkOrderId				:= tyBoardArrived2.tyData.sWorkOrdedId <> '';
				tyBoardArrived2.tyAvl.bBatchId			    	:= tyBoardArrived2.tyData.sBatchId <> '';

			END_IF

		END_IF

	END_IF

END_ACTION
```

#### Act_Background_SendBoardArrivedLane3.st - Do Not Change!!!
```iecst
(** 2021-08-01 **)
ACTION Act_Background_SendBoardArrivedLane3: //Send after our machine send out "StopTransport" message to upstream

	IF eStatus2 <> Error THEN
		IF tySServiceDescriptionRcv.tyData.tySupportedFeatures.bFeatureBoardTracking = TRUE AND p_tyParam.bFeatureBoardTracking AND bHandshakeDone THEN
			IF EDGEPOS(p_bUSHermesStopTransport3) THEN

				fHermesAddOneMsgSend(ADR(a_eMsgSend) , ADR(udiMsgSendBffr) , HermesMsgTypeBoardArrived3);

				tyBoardArrived3.tyData.sMachineId     	        := p_sMcId;
				tyBoardArrived3.tyData.iUpstreamLaneId    	    := p_tyHermesConfiguration.a_tyUSParam[2].iLaneID;
				tyBoardArrived3.tyData.sUpstreamInterfaceId     := p_tyHermesConfiguration.a_tyUSParam[2].sUpstreamInterfaceId;
				tyBoardArrived3.tyData.sMagazineId           	:= sMagazineId;
				tyBoardArrived3.tyData.iSlotId     	            := iSlotId;
				tyBoardArrived3.tyData.eBoadTransfer    	    := HermesTransferred;
				tyBoardArrived3.tyData.sBoardId     	        := p_tyUSBoardArrived3.tyData.sBoardId;
				tyBoardArrived3.tyData.sBoardIdCreatedBy     	:= p_tyUSBoardArrived3.tyData.sBoardIdCreatedBy;
				tyBoardArrived3.tyData.eFailedBoard				:= p_tyUSBoardArrived3.tyData.eFailedBoard;
				tyBoardArrived3.tyData.sProductTypeId			:= p_tyUSBoardArrived3.tyData.sProductTypeId;
				tyBoardArrived3.tyData.eFlippedBoard		  	:= p_tyUSBoardArrived3.tyData.eFlippedBoard;
				tyBoardArrived3.tyData.sTopBarcode				:= p_tyUSBoardArrived3.tyData.sTopBarcode;
				tyBoardArrived3.tyData.sBottomBarcode			:= p_tyUSBoardArrived3.tyData.sBottomBarcode;
				tyBoardArrived3.tyData.rLength					:= p_tyUSBoardArrived3.tyData.rLength;
				tyBoardArrived3.tyData.rWidth				    := p_tyUSBoardArrived3.tyData.rWidth;
				tyBoardArrived3.tyData.rThickness				:= p_tyUSBoardArrived3.tyData.rThickness;
				tyBoardArrived3.tyData.rConveyorSpeed		    := p_tyUSBoardArrived3.tyData.rConveyorSpeed;
				tyBoardArrived3.tyData.rTopClearanceHeight		:= p_tyUSBoardArrived3.tyData.rTopClearanceHeight;
				tyBoardArrived3.tyData.rBottomClearanceHeight	:= p_tyUSBoardArrived3.tyData.rBottomClearanceHeight;
				tyBoardArrived3.tyData.rWeight					:= p_tyUSBoardArrived3.tyData.rWeight;
				tyBoardArrived3.tyData.sWorkOrdedId             := p_tyUSBoardArrived3.tyData.sWorkOrderId;
				tyBoardArrived3.tyData.sBatchId                 := p_tyUSBoardArrived3.tyData.sBatchId;

			    tyBoardArrived3.tyAvl.bMachineId				:= tyBoardArrived3.tyData.sMachineId <> '';
		     	tyBoardArrived3.tyAvl.bUpstreamLaneId			:= tyBoardArrived3.tyData.iUpstreamLaneId <> 0;
		    	tyBoardArrived3.tyAvl.bUpstreamInterfaceId		:= tyBoardArrived3.tyData.sUpstreamInterfaceId <> '';
		    	tyBoardArrived3.tyAvl.bMagazineId		    	:= tyBoardArrived3.tyData.sMagazineId <> '';
		    	tyBoardArrived3.tyAvl.bSlotId				    := tyBoardArrived3.tyData.iSlotId <> 0;
		    	tyBoardArrived3.tyAvl.bBoardTransfer			:= TRUE;
				tyBoardArrived3.tyAvl.bBoardId					:= tyBoardArrived3.tyData.sBoardId <> '';
				tyBoardArrived3.tyAvl.bBoardIdCreatedBy			:= tyBoardArrived3.tyData.sBoardIdCreatedBy <> '';
				tyBoardArrived3.tyAvl.bFailedBoard				:= TRUE;
				tyBoardArrived3.tyAvl.bProductTypeId		  	:= tyBoardArrived3.tyData.sProductTypeId <> '';
				tyBoardArrived3.tyAvl.bFlippedBoard				:= TRUE;
				tyBoardArrived3.tyAvl.bTopBarcode			    := tyBoardArrived3.tyData.sTopBarcode <> '';
				tyBoardArrived3.tyAvl.bBottomBarcode		   	:= tyBoardArrived3.tyData.sBottomBarcode <> '';
				tyBoardArrived3.tyAvl.bLength				    := tyBoardArrived3.tyData.rLength <> 0;
				tyBoardArrived3.tyAvl.bWidth				  	:= (tyBoardArrived3.tyData.rWidth <> 0);
				tyBoardArrived3.tyAvl.bThickness			   	:= (tyBoardArrived3.tyData.rThickness <> 0);
				tyBoardArrived3.tyAvl.bConveyorSpeed		   	:= tyBoardArrived3.tyData.rConveyorSpeed <> 0;
				tyBoardArrived3.tyAvl.bTopClearanceHeight	    := (tyBoardArrived3.tyData.rTopClearanceHeight <> 0);
				tyBoardArrived3.tyAvl.bBottomClearanceHeight    := (tyBoardArrived3.tyData.rBottomClearanceHeight <> 0);
		    	tyBoardArrived3.tyAvl.bWeight				    := tyBoardArrived3.tyData.rWeight <> 0;
				tyBoardArrived3.tyAvl.bWorkOrderId				:= tyBoardArrived3.tyData.sWorkOrdedId <> '';
				tyBoardArrived3.tyAvl.bBatchId			    	:= tyBoardArrived3.tyData.sBatchId <> '';

			END_IF

		END_IF

	END_IF

END_ACTION
```

#### Act_Background_SendBoardArrivedLane4.st - Do Not Change!!!
```iecst
(** 2021-08-01 **)
ACTION Act_Background_SendBoardArrivedLane4: //Send after our machine send out "StopTransport" message to upstream

	IF eStatus2 <> Error THEN
		IF tySServiceDescriptionRcv.tyData.tySupportedFeatures.bFeatureBoardTracking = TRUE AND p_tyParam.bFeatureBoardTracking AND bHandshakeDone THEN
			IF EDGEPOS(p_bUSHermesStopTransport4) THEN

				fHermesAddOneMsgSend(ADR(a_eMsgSend) , ADR(udiMsgSendBffr) , HermesMsgTypeBoardArrived4);

				tyBoardArrived4.tyData.sMachineId     	        := p_sMcId;
				tyBoardArrived4.tyData.iUpstreamLaneId    	    := p_tyHermesConfiguration.a_tyUSParam[3].iLaneID;
				tyBoardArrived4.tyData.sUpstreamInterfaceId     := p_tyHermesConfiguration.a_tyUSParam[3].sUpstreamInterfaceId;
				tyBoardArrived4.tyData.sMagazineId           	:= sMagazineId;
				tyBoardArrived4.tyData.iSlotId     	            := iSlotId;
				tyBoardArrived4.tyData.eBoadTransfer    	    := HermesTransferred;
				tyBoardArrived4.tyData.sBoardId     	        := p_tyUSBoardArrived4.tyData.sBoardId;
				tyBoardArrived4.tyData.sBoardIdCreatedBy     	:= p_tyUSBoardArrived4.tyData.sBoardIdCreatedBy;
				tyBoardArrived4.tyData.eFailedBoard				:= p_tyUSBoardArrived4.tyData.eFailedBoard;
				tyBoardArrived4.tyData.sProductTypeId			:= p_tyUSBoardArrived4.tyData.sProductTypeId;
				tyBoardArrived4.tyData.eFlippedBoard		  	:= p_tyUSBoardArrived4.tyData.eFlippedBoard;
				tyBoardArrived4.tyData.sTopBarcode				:= p_tyUSBoardArrived4.tyData.sTopBarcode;
				tyBoardArrived4.tyData.sBottomBarcode			:= p_tyUSBoardArrived4.tyData.sBottomBarcode;
				tyBoardArrived4.tyData.rLength					:= p_tyUSBoardArrived4.tyData.rLength;
				tyBoardArrived4.tyData.rWidth				    := p_tyUSBoardArrived4.tyData.rWidth;
				tyBoardArrived4.tyData.rThickness				:= p_tyUSBoardArrived4.tyData.rThickness;
				tyBoardArrived4.tyData.rConveyorSpeed		    := p_tyUSBoardArrived4.tyData.rConveyorSpeed;
				tyBoardArrived4.tyData.rTopClearanceHeight		:= p_tyUSBoardArrived4.tyData.rTopClearanceHeight;
				tyBoardArrived4.tyData.rBottomClearanceHeight	:= p_tyUSBoardArrived4.tyData.rBottomClearanceHeight;
				tyBoardArrived4.tyData.rWeight					:= p_tyUSBoardArrived4.tyData.rWeight;
				tyBoardArrived4.tyData.sWorkOrdedId             := p_tyUSBoardArrived4.tyData.sWorkOrderId;
				tyBoardArrived4.tyData.sBatchId                 := p_tyUSBoardArrived4.tyData.sBatchId;

			    tyBoardArrived4.tyAvl.bMachineId				:= tyBoardArrived4.tyData.sMachineId <> '';
		     	tyBoardArrived4.tyAvl.bUpstreamLaneId			:= tyBoardArrived4.tyData.iUpstreamLaneId <> 0;
		    	tyBoardArrived4.tyAvl.bUpstreamInterfaceId		:= tyBoardArrived4.tyData.sUpstreamInterfaceId <> '';
		    	tyBoardArrived4.tyAvl.bMagazineId		    	:= tyBoardArrived4.tyData.sMagazineId <> '';
		    	tyBoardArrived4.tyAvl.bSlotId				    := tyBoardArrived4.tyData.iSlotId <> 0;
		    	tyBoardArrived4.tyAvl.bBoardTransfer			:= TRUE;
				tyBoardArrived4.tyAvl.bBoardId					:= tyBoardArrived4.tyData.sBoardId <> '';
				tyBoardArrived4.tyAvl.bBoardIdCreatedBy			:= tyBoardArrived4.tyData.sBoardIdCreatedBy <> '';
				tyBoardArrived4.tyAvl.bFailedBoard				:= TRUE;
				tyBoardArrived4.tyAvl.bProductTypeId		  	:= tyBoardArrived4.tyData.sProductTypeId <> '';
				tyBoardArrived4.tyAvl.bFlippedBoard				:= TRUE;
				tyBoardArrived4.tyAvl.bTopBarcode			    := tyBoardArrived4.tyData.sTopBarcode <> '';
				tyBoardArrived4.tyAvl.bBottomBarcode		   	:= tyBoardArrived4.tyData.sBottomBarcode <> '';
				tyBoardArrived4.tyAvl.bLength				    := tyBoardArrived4.tyData.rLength <> 0;
				tyBoardArrived4.tyAvl.bWidth				  	:= (tyBoardArrived4.tyData.rWidth <> 0);
				tyBoardArrived4.tyAvl.bThickness			   	:= (tyBoardArrived4.tyData.rThickness <> 0);
				tyBoardArrived4.tyAvl.bConveyorSpeed		   	:= tyBoardArrived4.tyData.rConveyorSpeed <> 0;
				tyBoardArrived4.tyAvl.bTopClearanceHeight	    := (tyBoardArrived4.tyData.rTopClearanceHeight <> 0);
				tyBoardArrived4.tyAvl.bBottomClearanceHeight    := (tyBoardArrived4.tyData.rBottomClearanceHeight <> 0);
		    	tyBoardArrived4.tyAvl.bWeight				    := tyBoardArrived4.tyData.rWeight <> 0;
				tyBoardArrived4.tyAvl.bWorkOrderId				:= tyBoardArrived4.tyData.sWorkOrdedId <> '';
				tyBoardArrived4.tyAvl.bBatchId			    	:= tyBoardArrived4.tyData.sBatchId <> '';

			END_IF

		END_IF

	END_IF

END_ACTION
```

#### Act_Background_SendBoardDepartedLane1.st - Do Not Change!!!
```iecst
(** 2021-08-01 **)
ACTION Act_Background_SendBoardDepartedLane1: //Send after our machine send out "TransportFinished" message to downstream

	IF eStatus2 <> Error THEN
		IF tySServiceDescriptionRcv.tyData.tySupportedFeatures.bFeatureBoardTracking = TRUE AND p_tyParam.bFeatureBoardTracking AND bHandshakeDone THEN
			IF EDGEPOS(p_bDSHermesTransportFinished1) THEN

				fHermesAddOneMsgSend(ADR(a_eMsgSend) , ADR(udiMsgSendBffr) , HermesMsgTypeBoardDeparted1);

				tyBoardDeparted1.tyData.sMachineId     	        := p_sMcId;
			    tyBoardDeparted1.tyData.iDownstreamLaneId    	:= p_tyHermesConfiguration.a_tyDSParam[0].iLaneID;
			    tyBoardDeparted1.tyData.sDownstreamInterfaceId  := p_tyHermesConfiguration.a_tyDSParam[0].sDownstreamInterfaceId;
                tyBoardDeparted1.tyData.sMagazineId           	:= sMagazineId;
		    	tyBoardDeparted1.tyData.iSlotId     	        := iSlotId;
		    	tyBoardDeparted1.tyData.eBoadTransfer    	    := p_eBoardTransfer1;
	            tyBoardDeparted1.tyData.sBoardId     	        := p_tyDSBoardDeparted1.tyData.sBoardId;
		    	tyBoardDeparted1.tyData.sBoardIdCreatedBy     	:= p_tyDSBoardDeparted1.tyData.sBoardIdCreatedBy;
		    	tyBoardDeparted1.tyData.eFailedBoard			:= p_tyDSBoardDeparted1.tyData.eFailedBoard;
				tyBoardDeparted1.tyData.sProductTypeId			:= p_tyDSBoardDeparted1.tyData.sProductTypeId;
				tyBoardDeparted1.tyData.eFlippedBoard			:= p_tyDSBoardDeparted1.tyData.eFlippedBoard;
				tyBoardDeparted1.tyData.sTopBarcode				:= p_tyDSBoardDeparted1.tyData.sTopBarcode;
				tyBoardDeparted1.tyData.sBottomBarcode			:= p_tyDSBoardDeparted1.tyData.sBottomBarcode;
				tyBoardDeparted1.tyData.rLength					:= p_tyDSBoardDeparted1.tyData.rLength;
				tyBoardDeparted1.tyData.rWidth				    := p_tyDSBoardDeparted1.tyData.rWidth;
				tyBoardDeparted1.tyData.rThickness				:= p_tyDSBoardDeparted1.tyData.rThickness;
				tyBoardDeparted1.tyData.rConveyorSpeed		    := p_tyDSBoardDeparted1.tyData.rConveyorSpeed;
				tyBoardDeparted1.tyData.rTopClearanceHeight		:= p_tyDSBoardDeparted1.tyData.rTopClearanceHeight;
				tyBoardDeparted1.tyData.rBottomClearanceHeight	:= p_tyDSBoardDeparted1.tyData.rBottomClearanceHeight;
				tyBoardDeparted1.tyData.rWeight					:= p_tyDSBoardDeparted1.tyData.rWeight;
				tyBoardDeparted1.tyData.sWorkOrdedId            := p_tyDSBoardDeparted1.tyData.sWorkOrderId;
				tyBoardDeparted1.tyData.sBatchId                := p_tyDSBoardDeparted1.tyData.sBatchId;

			    tyBoardDeparted1.tyAvl.bMachineId				:= tyBoardDeparted1.tyData.sMachineId <> '';
		     	tyBoardDeparted1.tyAvl.bDownstreamLaneId		:= tyBoardDeparted1.tyData.iDownstreamLaneId <> 0;
		    	tyBoardDeparted1.tyAvl.bDownstreamInterfaceId	:= tyBoardDeparted1.tyData.sDownstreamInterfaceId <> '';
		    	tyBoardDeparted1.tyAvl.bMagazineId		    	:= tyBoardDeparted1.tyData.sMagazineId <> '';
		    	tyBoardDeparted1.tyAvl.bSlotId				    := tyBoardDeparted1.tyData.iSlotId <> 0;
		    	tyBoardDeparted1.tyAvl.bBoardTransfer		    := TRUE;
				tyBoardDeparted1.tyAvl.bBoardId					:= tyBoardDeparted1.tyData.sBoardId <> '';
				tyBoardDeparted1.tyAvl.bBoardIdCreatedBy		:= tyBoardDeparted1.tyData.sBoardIdCreatedBy <> '';
				tyBoardDeparted1.tyAvl.bFailedBoard				:= TRUE;
				tyBoardDeparted1.tyAvl.bProductTypeId		   	:= tyBoardDeparted1.tyData.sProductTypeId <> '';
				tyBoardDeparted1.tyAvl.bFlippedBoard			:= TRUE;
				tyBoardDeparted1.tyAvl.bTopBarcode			    := tyBoardDeparted1.tyData.sTopBarcode <> '';
				tyBoardDeparted1.tyAvl.bBottomBarcode		    := tyBoardDeparted1.tyData.sBottomBarcode <> '';
				tyBoardDeparted1.tyAvl.bLength				    := tyBoardDeparted1.tyData.rLength <> 0;
				tyBoardDeparted1.tyAvl.bWidth				    := (tyBoardDeparted1.tyData.rWidth <> 0);
				tyBoardDeparted1.tyAvl.bThickness			    := (tyBoardDeparted1.tyData.rThickness <> 0);
				tyBoardDeparted1.tyAvl.bConveyorSpeed		    := tyBoardDeparted1.tyData.rConveyorSpeed <> 0;
				tyBoardDeparted1.tyAvl.bTopClearanceHeight	    := (tyBoardDeparted1.tyData.rTopClearanceHeight <> 0);
				tyBoardDeparted1.tyAvl.bBottomClearanceHeight	:= (tyBoardDeparted1.tyData.rBottomClearanceHeight <> 0);
		    	tyBoardDeparted1.tyAvl.bWeight				    := tyBoardDeparted1.tyData.rWeight <> 0;
				tyBoardDeparted1.tyAvl.bWorkOrderId				:= tyBoardDeparted1.tyData.sWorkOrdedId <> '';
				tyBoardDeparted1.tyAvl.bBatchId			    	:= tyBoardDeparted1.tyData.sBatchId <> '';

			END_IF

		END_IF

	END_IF

END_ACTION
```

#### Act_Background_SendBoardDepartedLane2.st - Do Not Change!!!
```iecst
(** 2021-08-01 **)
ACTION Act_Background_SendBoardDepartedLane2: //Send after our machine send out "TransportFinished" message to downstream

	IF eStatus2 <> Error THEN
		IF tySServiceDescriptionRcv.tyData.tySupportedFeatures.bFeatureBoardTracking = TRUE AND p_tyParam.bFeatureBoardTracking AND bHandshakeDone THEN
			IF EDGEPOS(p_bDSHermesTransportFinished2) THEN

				fHermesAddOneMsgSend(ADR(a_eMsgSend) , ADR(udiMsgSendBffr) , HermesMsgTypeBoardDeparted2);

				tyBoardDeparted2.tyData.sMachineId     	        := p_sMcId;
			    tyBoardDeparted2.tyData.iDownstreamLaneId    	:= p_tyHermesConfiguration.a_tyDSParam[1].iLaneID;
			    tyBoardDeparted2.tyData.sDownstreamInterfaceId  := p_tyHermesConfiguration.a_tyDSParam[1].sDownstreamInterfaceId;
                tyBoardDeparted2.tyData.sMagazineId           	:= sMagazineId;
		    	tyBoardDeparted2.tyData.iSlotId     	        := iSlotId;
		    	tyBoardDeparted2.tyData.eBoadTransfer    	    := p_eBoardTransfer2;
	            tyBoardDeparted2.tyData.sBoardId     	        := p_tyDSBoardDeparted2.tyData.sBoardId;
		    	tyBoardDeparted2.tyData.sBoardIdCreatedBy     	:= p_tyDSBoardDeparted2.tyData.sBoardIdCreatedBy;
		    	tyBoardDeparted2.tyData.eFailedBoard			:= p_tyDSBoardDeparted2.tyData.eFailedBoard;
				tyBoardDeparted2.tyData.sProductTypeId			:= p_tyDSBoardDeparted2.tyData.sProductTypeId;
				tyBoardDeparted2.tyData.eFlippedBoard			:= p_tyDSBoardDeparted2.tyData.eFlippedBoard;
				tyBoardDeparted2.tyData.sTopBarcode				:= p_tyDSBoardDeparted2.tyData.sTopBarcode;
				tyBoardDeparted2.tyData.sBottomBarcode			:= p_tyDSBoardDeparted2.tyData.sBottomBarcode;
				tyBoardDeparted2.tyData.rLength					:= p_tyDSBoardDeparted2.tyData.rLength;
				tyBoardDeparted2.tyData.rWidth				    := p_tyDSBoardDeparted2.tyData.rWidth;
				tyBoardDeparted2.tyData.rThickness				:= p_tyDSBoardDeparted2.tyData.rThickness;
				tyBoardDeparted2.tyData.rConveyorSpeed		    := p_tyDSBoardDeparted2.tyData.rConveyorSpeed;
				tyBoardDeparted2.tyData.rTopClearanceHeight		:= p_tyDSBoardDeparted2.tyData.rTopClearanceHeight;
				tyBoardDeparted2.tyData.rBottomClearanceHeight	:= p_tyDSBoardDeparted2.tyData.rBottomClearanceHeight;
				tyBoardDeparted2.tyData.rWeight					:= p_tyDSBoardDeparted2.tyData.rWeight;
				tyBoardDeparted2.tyData.sWorkOrdedId            := p_tyDSBoardDeparted2.tyData.sWorkOrderId;
				tyBoardDeparted2.tyData.sBatchId                := p_tyDSBoardDeparted2.tyData.sBatchId;

			    tyBoardDeparted2.tyAvl.bMachineId				:= tyBoardDeparted2.tyData.sMachineId <> '';
		     	tyBoardDeparted2.tyAvl.bDownstreamLaneId		:= tyBoardDeparted2.tyData.iDownstreamLaneId <> 0;
		    	tyBoardDeparted2.tyAvl.bDownstreamInterfaceId	:= tyBoardDeparted2.tyData.sDownstreamInterfaceId <> '';
		    	tyBoardDeparted2.tyAvl.bMagazineId		    	:= tyBoardDeparted2.tyData.sMagazineId <> '';
		    	tyBoardDeparted2.tyAvl.bSlotId				    := tyBoardDeparted2.tyData.iSlotId <> 0;
		    	tyBoardDeparted2.tyAvl.bBoardTransfer		    := TRUE;
				tyBoardDeparted2.tyAvl.bBoardId					:= tyBoardDeparted2.tyData.sBoardId <> '';
				tyBoardDeparted2.tyAvl.bBoardIdCreatedBy		:= tyBoardDeparted2.tyData.sBoardIdCreatedBy <> '';
				tyBoardDeparted2.tyAvl.bFailedBoard				:= TRUE;
				tyBoardDeparted2.tyAvl.bProductTypeId		   	:= tyBoardDeparted2.tyData.sProductTypeId <> '';
				tyBoardDeparted2.tyAvl.bFlippedBoard			:= TRUE;
				tyBoardDeparted2.tyAvl.bTopBarcode			    := tyBoardDeparted2.tyData.sTopBarcode <> '';
				tyBoardDeparted2.tyAvl.bBottomBarcode		    := tyBoardDeparted2.tyData.sBottomBarcode <> '';
				tyBoardDeparted2.tyAvl.bLength				    := tyBoardDeparted2.tyData.rLength <> 0;
				tyBoardDeparted2.tyAvl.bWidth				    := (tyBoardDeparted2.tyData.rWidth <> 0);
				tyBoardDeparted2.tyAvl.bThickness			    := (tyBoardDeparted2.tyData.rThickness <> 0);
				tyBoardDeparted2.tyAvl.bConveyorSpeed		    := tyBoardDeparted2.tyData.rConveyorSpeed <> 0;
				tyBoardDeparted2.tyAvl.bTopClearanceHeight	    := (tyBoardDeparted2.tyData.rTopClearanceHeight <> 0);
				tyBoardDeparted2.tyAvl.bBottomClearanceHeight	:= (tyBoardDeparted2.tyData.rBottomClearanceHeight <> 0);
		    	tyBoardDeparted2.tyAvl.bWeight				    := tyBoardDeparted2.tyData.rWeight <> 0;
				tyBoardDeparted2.tyAvl.bWorkOrderId				:= tyBoardDeparted2.tyData.sWorkOrdedId <> '';
				tyBoardDeparted2.tyAvl.bBatchId			    	:= tyBoardDeparted2.tyData.sBatchId <> '';

			END_IF

		END_IF

	END_IF

END_ACTION
```
